// TIA Portal project "Vessel Recycle System 1 Rev1.0" (V14)

(* hardware
DEVICE "S71500/ET200MP station_1"  S7-1500 station
   slot 0: "Rail_0"  Rack  6ES7 590-1***0-0AA0
   slot 0: "PM 70W 120/230VAC"  PM 70W 120/230VAC  6EP1332-4BA00
   slot 1: "PLC_1"  CPU 1511-1 PN  6ES7 511-1AK01-0AB0  V2.0
      slot 3: "CPU display_1"  6ES7591-1AA00-0AA0
DEVICE "ET 200SP station_1"  ET 200SP-Station
   slot 0: "Rack_0"  Rack  6ES5 710-8MAx1
   slot 0: "IO device_1"  IM 155-6 PN BA  6ES7 155-6AR00-0AN0  V3.2
   slot 1: "DI 8x24VDC BA_1"  DI 8x24VDC BA  6ES7 131-6BF00-0AA0  V1.0
      slot 1: "DI 8x24VDC BA_1"  DI 8x24VDC BA
   slot 2: "DI 8x24VDC BA_2"  DI 8x24VDC BA  6ES7 131-6BF00-0AA0  V1.0
      slot 1: "DI 8x24VDC BA_2"  DI 8x24VDC BA
   slot 3: "DQ 8x24VDC/0.5A BA_1"  DQ 8x24VDC/0.5A BA  6ES7 132-6BF00-0AA0  V1.0
      slot 1: "DQ 8x24VDC/0.5A BA_1"  DQ 8x24VDC/0.5A BA
   slot 4: "DQ 8x24VDC/0.5A BA_2"  DQ 8x24VDC/0.5A BA  6ES7 132-6BF00-0AA0  V1.0
      slot 1: "DQ 8x24VDC/0.5A BA_2"  DQ 8x24VDC/0.5A BA
   slot 5: "DQ 8x24VDC/0.5A BA_3"  DQ 8x24VDC/0.5A BA  6ES7 132-6BF00-0AA0  V1.0
      slot 1: "DQ 8x24VDC/0.5A BA_3"  DQ 8x24VDC/0.5A BA
   slot 6: "Server module_1"  Server module  6ES7 193-6PA00-0AA0  V1.1
      slot 1: "Server module_1"  Server module
   slot 127: "BA 2xRJ45"  BA 2xRJ45  6ES7 193-6AR00-0AA0  V0.0
      slot 1: "Port_1"  6ES7 193-6AR00-0AA0  V0.0
      slot 2: "Port_2"  6ES7 193-6AR00-0AA0  V0.0
DEVICE "SCALANCE XB-200"  SCALANCE X-Station
   slot 0: "SCALANCE X rack"  Rail
   slot 0: "Switch_1"  SCALANCE XB208  6GK5 208-0BA00-2AB2  V1.2
DEVICE "HMI_1"  TP1200 Comfort
   slot 0: "TP1200 Comfort"  TP1200 Comfort  6AV2 124-0MC01-0AX0  14.0.0.0
   slot 1: "HMI_RT_1"  TP1200 Comfort  6AV2 124-0MC01-0AX0  14.0.0.0
   slot 5: "HMI_1.IE_CP_1"  PROFINET Interface  14.0.0.0
      slot 1: "PROFINET Interface_1"  PROFINET Interface
         slot 1: "Port_1"  Port
         slot 2: "Port_2"  Port
   slot 7: "HMI_1.MPI/DP_CP_1"  MPI/DP Interface  14.0.0.0
DEVICE "GSD device_1"  GSD.Device.PN
   slot 0: "Rack"  Rack  V1.0
   slot 0: "vr1pump1"  Standard, no PDev  6GK1 953-0CA00  Z1.0
      slot 0: "Standard, no PDev"  Standard, no PDev
      slot 1: "Interface"  Interface
         slot 1: "Port_1"  Port
   slot 1: " 128 bytes I_1"  128 bytes I  1.0
      slot 0: " 128 bytes I"  128 bytes I
   slot 2: " 128 bytes O_1"  128 bytes O  1.0
      slot 0: " 128 bytes O"  128 bytes O
DEVICE "GSD device_2"  GSD.Device.PN
   slot 0: "Rack"  Rack  V1.0
   slot 0: "vr1pump2"  Standard, no PDev  6GK1 953-0CA00  Z1.0
      slot 0: "Standard, no PDev"  Standard, no PDev
      slot 1: "Interface"  Interface
         slot 1: "Port_1"  Port
   slot 1: " 128 bytes I_1"  128 bytes I  1.0
      slot 0: " 128 bytes I"  128 bytes I
   slot 2: " 128 bytes O_1"  128 bytes O  1.0
      slot 0: " 128 bytes O"  128 bytes O
*)

// ===== PLC "PLC_1"  CPU 1511-1 PN =====

VAR_GLOBAL   // PLC tag table "Default tag table"
   "System_Byte" AT %MB1 : Byte;
   "FirstScan" AT %M1.0 : Bool;
   "DiagStatusUpdate" AT %M1.1 : Bool;
   "AlwaysTRUE" AT %M1.2 : Bool;
   "AlwaysFALSE" AT %M1.3 : Bool;
   "Clock_Byte" AT %MB0 : Byte;
   "Clock_10Hz" AT %M0.0 : Bool;
   "Clock_5Hz" AT %M0.1 : Bool;
   "Clock_2.5Hz" AT %M0.2 : Bool;
   "Clock_2Hz" AT %M0.3 : Bool;
   "Clock_1.25Hz" AT %M0.4 : Bool;
   "Clock_1Hz" AT %M0.5 : Bool;
   "Clock_0.625Hz" AT %M0.6 : Bool;
   "Clock_0.5Hz" AT %M0.7 : Bool;
END_VAR

VAR_GLOBAL   // PLC tag table "General Tags"
   "Safety_Relay_Trip" AT %I0.0 : Bool;
   "spare_%I0.3" AT %I0.3 : Bool;
   "UM_HI_Level_SW" AT %I0.6 : Bool;
   "spare_%I0.7" AT %I0.7 : Bool;
   "spare_%Q0.0" AT %Q0.0 : Bool;
   "spare_%Q0.1" AT %Q0.1 : Bool;
   "spare_%Q2.2" AT %Q2.2 : Bool;
   "Buzzer" AT %Q2.5 : Bool;
   "Green_Light" AT %Q2.6 : Bool;
   "Red_Light" AT %Q2.7 : Bool;
   "spare_%Q1.2" AT %Q1.2 : Bool;
   "spare_%Q1.3" AT %Q1.3 : Bool;
   "spare_%Q1.4" AT %Q1.4 : Bool;
   "spare_%Q1.5" AT %Q1.5 : Bool;
   "spare_%Q1.6" AT %Q1.6 : Bool;
   "spare_%Q1.7" AT %Q1.7 : Bool;
   "spare_%I1.6" AT %I1.6 : Bool;
   "spare_%I1.7" AT %I1.7 : Bool;
   "spare_%Q0.2" AT %Q0.2 : Bool;
   "spare_%Q0.3" AT %Q0.3 : Bool;
END_VAR

VAR_GLOBAL   // PLC tag table "Station 1"
   "S1_Start_PB" AT %I0.1 : Bool;
   "S1_Stop_PB" AT %I0.2 : Bool;
   "Safety_Lock1_Engaged" AT %I1.0 : Bool;
   "Safety_Key1_Inserted" AT %I1.1 : Bool;
   "Estop1_PB_Active" AT %I1.4 : Bool;
   "S1_Valve" AT %Q0.4 : Bool;
   "Safety_Lock1_Open" AT %Q0.5 : Bool;
   "Pmp1_Permissive" AT %Q1.0 : Bool;
   "S1_Start_Light" AT %Q2.0 : Bool;
   "S1_Stop_Light" AT %Q2.1 : Bool;
END_VAR

VAR_GLOBAL   // PLC tag table "Station 2"
   "S2_Start_PB" AT %I0.4 : Bool;
   "S2_Stop_PB" AT %I0.5 : Bool;
   "Safety_Lock2_Engaged" AT %I1.2 : Bool;
   "Safety_Key2_Inserted" AT %I1.3 : Bool;
   "Estop2_PB_Active" AT %I1.5 : Bool;
   "S2_Valve" AT %Q0.6 : Bool;
   "Safety_Lock2_Open" AT %Q0.7 : Bool;
   "Pmp2_Permissive" AT %Q1.1 : Bool;
   "S2_Start_Light" AT %Q2.3 : Bool;
   "S2_Stop_Light" AT %Q2.4 : Bool;
END_VAR

TYPE "UDT_MDrive_PQW"
   STRUCT
      Acc : UDInt;   // A
      Dec : UDInt;   // D
      TS : UDInt;   // TS
      V_Init : UDInt;   // VI
      V_Max : UDInt;   // VM
      C1 : DInt;   // C1
      C2 : DInt;   // C2
      HT : DInt;   // HT
      MoveABS : DInt;   // MA
      MoveRel : DInt;   // MR
      Slew : DInt;   // SL
      SetPosition : DInt;   // P
      MT : DInt;   // MT
      MS : UInt;   // MS
      SetError : UInt;   // ER
      AO : UInt;   // AO
      AS : USInt;   // AS
      HC : USInt;   // HC
      OT : USInt;   // OT
      RC : USInt;   // RC
      TQ : USInt;   // TQ
      HM : USInt;   // HM
      HI : USInt;   // HI
      DriveEnable : USInt;   // DriveEnable
      EncoderEnable : USInt;   // EncoderEnable
      TD : USInt;   // TD
      Esc : USInt;   // Esc
      CF : USInt;   // CF
      R9_R10 : Struct
         Reg9 : Bool;
         Bit1 : Bool;
         Bit2 : Bool;
         Bit3 : Bool;
         Bit4 : Bool;
         Bit5 : Bool;
         Bit6 : Bool;
         Bit7 : Bool;
         Reg10 : Bool;
         Bit8 : Bool;
         Bit9 : Bool;
         Bit10 : Bool;
         Bit11 : Bool;
         Bit12 : Bool;
         Bit13 : Bool;
         Bit14 : Bool;
      END_STRUCT;
      R11 : Struct
         Reg11 : Bool;
         Bit1 : Bool;
         Bit2 : Bool;
         Bit3 : Bool;
         Bit4 : Bool;
         Bit5 : Bool;
         Bit6 : Bool;
         Bit7 : Bool;
      END_STRUCT;
      Unused_1 : String[28];
      R1_R38 : Struct
         Dummy_Bit0 : Bool;
         Dummy_Bit1 : Bool;
         Dummy_Bit2 : Bool;
         Dummy_Bit3 : Bool;
         Dummy_Bit4 : Bool;
         Dummy_Bit5 : Bool;
         Dummy_Bit6 : Bool;
         Dummy_Bit7 : Bool;
         Reg1 : Bool;
         Reg2 : Bool;
         Reg3 : Bool;
         Reg4 : Bool;
         Reg5 : Bool;
         Reg6 : Bool;
         Reg7 : Bool;
         Reg8 : Bool;
         Reg9 : Bool;
         Reg10 : Bool;
         Reg11 : Bool;
         Reg12 : Bool;
         Reg13 : Bool;
         Reg14 : Bool;
         Reg15 : Bool;
         Reg16 : Bool;
         Reg17 : Bool;
         Reg18 : Bool;
         Reg19 : Bool;
         Reg20 : Bool;
         Reg21 : Bool;
         Reg22 : Bool;
         Reg23 : Bool;
         Reg24 : Bool;
         Reg25 : Bool;
         Reg26 : Bool;
         Reg27 : Bool;
         Reg28 : Bool;
         Reg32 : Bool;
         Reg33 : Bool;
         Reg38 : Bool;
         Dummy_Bit8 : Bool;
         Dummy_Bit9 : Bool;
         Dummy_Bit10 : Bool;
         Dummy_Bit11 : Bool;
         Dummy_Bit12 : Bool;
         Dummy_Bit13 : Bool;
         Dummy_Bit14 : Bool;
         Dummy_Bit15 : Bool;
         Dummy_Bit16 : Bool;
      END_STRUCT;
      Unused_2 : Array[0..17] of Byte;
   END_STRUCT;
END_TYPE

TYPE "UDT_MDrive_PIW"
   STRUCT
      Acc : UDInt;   // A
      Dec : UDInt;   // D
      TS : UDInt;   // TS
      V_Init : UDInt;   // VI
      V_Max : UDInt;   // VM
      C1 : DInt;   // C1
      C2 : DInt;   // C2
      LL : DInt;   // LL
      V : DInt;   // V
      PC : DInt;   // PC
      MS : DInt;   // MS
      Position : DInt;   // P
      AO : UInt;   // AO
      Dummy_Int : UInt;   // Dummy_Int
      AF : UInt;   // AF
      Error : UInt;   // ER
      I5 : UInt;   // I5
      AS : USInt;   // AS
      HC : USInt;   // HC
      Inputs : USInt;   // IN
      RC : USInt;   // RC
      TQ : USInt;   // TQ
      "OF" : USInt;   // OF
      TE : USInt;   // TE
      DriveEnable : USInt;   // DriveEnable
      EncoderEnable : USInt;   // EncoderEnable
      TD : USInt;   // TD
      MV : USInt;   // MV
      MP : USInt;   // MP
      VC : USInt;   // VC
      ST : USInt;   // ST
      LR : USInt;   // LR
      Dummy_Byte : USInt;
      Unused : Array[0..52] of Byte;
   END_STRUCT;
END_TYPE

TYPE "UDT_MDrive_Data"
   STRUCT
      Target_Position : DInt;   // Input
      Current_Position : DInt := 0;   // Output
      Slew : Struct   // Input
         Fwd : Bool;   // Input
         Rev : Bool;   // Input
         Speed : Real;   // Input
      END_STRUCT;
      State : Struct   // Output
         IsMoving : Bool;   // Output
         IsHomed : Bool;   // Output
         OnPosition : Bool;   // Output
      END_STRUCT;
      ErrorCode : UInt;   // Output
      Inputs : Array[0..7] of Bool;   // Output
      HomeSensor : Bool;   // Output
      Reset : Bool;   // Output
      CMD_Trigger : Struct   // Input
         MoveAbs : Bool;   // Trigger new MA command
         MoveRel : Bool;   // Trigger new MR command
         Slew : Bool;   // Trigger new SL command
         Homing : Bool;   // Trigger new HM command ( Homing )
         SetPos : Bool;   // Trigger new Position
      END_STRUCT;
      CMD_Busy : Bool;   // Output
   END_STRUCT;
END_TYPE

TYPE "UDT_MDrive_Settings"
   STRUCT
      ScaleMax : DInt;
      ScaleMin : DInt;
      MaxSpeed : DInt;
      MinSpeed : DInt;
   END_STRUCT;
END_TYPE

TYPE "UDT_HMI_MDrive"
   STRUCT
      Slew : Struct   // Input
         Fwd : Bool;   // Input
         Rev : Bool;   // Input
         Speed : Real;   // Input
      END_STRUCT;
      State : Struct   // Output
         IsMoving : Bool;   // Output
         IsHomed : Bool;   // Output
         OnPosition : Bool;   // Output
      END_STRUCT;
      Drive_State : USInt;   // Output
      ErrorCode : UInt;   // Output
   END_STRUCT;
END_TYPE

DATA_BLOCK "Setup_Data"   // DB2
{ S7_Optimized_Access := 'TRUE' }
VERSION : 0.1
   VAR
      Estop_Active : Bool;
      Buzzer_Reset : Bool;
   END_VAR
   VAR RETAIN
      Total_Waste_Drum_Volume : Real;
      Waste_Drum_Volume : Real := 100.0;
      Waste_Drum_Percent_Volume : Real;
   END_VAR
   VAR
      Waste_Container_Reset : Bool;
      Waste_Container_Interlock : Bool;
      Waste_Container_Alarm_Level : Int := 0;
      Waste_Container_Alarm_SP : Real := 80.0;
      Waste_Container_Interlock_Level : Real := 90.0;
      Waste_Rad_Level : Real;
   END_VAR
   VAR RETAIN
      Waste_Rad_High_Alarm : Real := 100.0;
   END_VAR
   VAR
      Waste_Rad_Alarm : Bool;
   END_VAR
   VAR RETAIN
      System_Version : String := 'VRS1 Ver 1.0';
   END_VAR
BEGIN
END_DATA_BLOCK

DATA_BLOCK "Discrete_Alarm_Source_DB"   // DB20
{ S7_Optimized_Access := 'TRUE' }
VERSION : 0.1
// stored: InstanceOfName Discrete_Alarm_Source
"Discrete_Alarm_Source"
BEGIN
END_DATA_BLOCK

// folder: Station 1 Data Blocks

DATA_BLOCK "S1_HMI_DB"   // DB1
{ S7_Optimized_Access := 'TRUE' }
VERSION : 0.1
// stored: InstanceOfName Station_HMI
"Station_HMI"
BEGIN
END_DATA_BLOCK

DATA_BLOCK "S1_Auto_Mode_Setpoints"   // DB3
{ S7_Optimized_Access := 'TRUE' }
VERSION : 0.1
   VAR RETAIN
      Pump_Remove_Full_Speed : Real := 300.0;
      Ramp_Remove_Step : Int := 1;
      Ramp_Remove_Time : Time := T#500MS;
      Pump_Drain_Full_Speed : Real := 475.0;
      Ramp_Drain_Step : Int := 1;
      Ramp_Drain_Time : Time := T#500MS;
      Pump_Rinse_Full_Speed : Real := 425.0;
      Ramp_Rinse_Step : Int := 1;
      Ramp_Rinse_Time : Time := T#500MS;
      Run_Remove_Time : Time := T#1M_3S;
      Run_Drain_Time : Time := T#27S;
      Run_Rinse_Time : Time := T#19S;
      Number_of_Rinses : Int := 3;
      Use_RAD_CTRL : Bool := FALSE;
      Rinse_to_RAD_Level : Real := 50.0;
   END_VAR
BEGIN
END_DATA_BLOCK

DATA_BLOCK "S1_General_Setup"   // DB6
{ S7_Optimized_Access := 'TRUE' }
VERSION : 0.1
   VAR
      Manual_Mode : Bool;
      MM_Run_Enable : Bool;
      Auto_Run_Enable : Bool;
      Man_Speed_SP : Real;
      MM_Pump_Slew_PB : Bool;
      MM_Pump_Dir_SW_FWD : Bool;
      MM_Pump_Dir_SW_REV : Bool;
      MM_Valve_Dir_SW : Bool;
      MM_Feedback_RPM : Real;
      Auto_Process_Complete : Bool;
      Auto_Process_Complete_Trig : Bool;
      Manual_Mode_Permissive : Bool;
      Door_Lock_Bypass : Bool;
      Water_Supply_Interlock : Bool;
      Pump_Encoder_Run : Bool;
      Vessel_Rad_Level : Real;
   END_VAR
   VAR RETAIN
      Vessel_Alarm_Level : Real := 100.0;
   END_VAR
   VAR
      Pump_Rad_Level : Real;
   END_VAR
   VAR RETAIN
      Pump_Alarm_Level : Real := 100.0;
   END_VAR
   VAR
      Rad_Lock_Bypass : Bool;
      Rad_Lock : Bool;
   END_VAR
   VAR RETAIN
      Leave_Manual_Screen : Bool;
      Container_Water_Supply_Volume : Real := 3.0;
      Total_Water_Supply_Volume : Real;
      Total_from_Water_Supply_Volume : Real;
      Water_Supply_Interlock_Level : Real := 3.0;
   END_VAR
   VAR
      Total_Water_Supply_Percent : Real;
   END_VAR
   VAR RETAIN
      Total_to_Waste_Volume : Real;
   END_VAR
   VAR
      Pump_Factor : Real := 1.0;
      Pump_Stroke_Volume : Real := 0.192;
      Water_Supply_Alarm_Level : Int;
      Water_Supply_Alarm_SP : Real := 20.0;
      MM_Pump_Feedback : Real;
      Auto_Pump_Feedback_Vel : Real;
      Auto_Pump_Feedback_En : DInt;
      Auto_Pump_Running : Bool;
      Pump_Feedback : Real;
      New_Waste_Container : Bool;
      New_Water_Container : Bool;
      Level_Interlock : Bool;
      Pump_Error_Code : UInt;
      Pump_Error_Bit : Bool;
      MM_Pump_Error_Code : UInt;
      MM_Pump_Error_Bit : Bool;
   END_VAR
BEGIN
END_DATA_BLOCK

DATA_BLOCK "S1_Automated_Run_DB"   // DB7
{ S7_Optimized_Access := 'TRUE' }
VERSION : 0.1
// stored: InstanceOfName Automated_Run
"Automated_Run"
BEGIN
END_DATA_BLOCK

DATA_BLOCK "S1_ Door_Lock_Control_DB"   // DB9
{ S7_Optimized_Access := 'TRUE' }
VERSION : 0.1
// stored: InstanceOfName Door_Lock_Control
"Door_Lock_Control"
BEGIN
END_DATA_BLOCK

DATA_BLOCK "S1_Interlocks_DB"   // DB10
{ S7_Optimized_Access := 'TRUE' }
VERSION : 0.1
// stored: InstanceOfName Interlocks
"Interlocks"
BEGIN
END_DATA_BLOCK

DATA_BLOCK "Manual_Run_S1_DB"   // DB23
{ S7_Optimized_Access := 'TRUE' }
VERSION : 0.1
// stored: InstanceOfName Manual_ Run
"Manual_ Run"
BEGIN
END_DATA_BLOCK

// folder: Station 1 Data Blocks/Pump 1 Data Blocks

DATA_BLOCK "Pmp1_MM_HMI_DB"   // DB5
{ S7_Optimized_Access := 'TRUE' }
VERSION : 0.1
// stored: InstanceOfName Pump_HMI
"Pump_HMI"
BEGIN
END_DATA_BLOCK

DATA_BLOCK "Pmp1_Auto_HMI_DB"   // DB13
{ S7_Optimized_Access := 'TRUE' }
VERSION : 0.1
// stored: InstanceOfName Pump_HMI
"Pump_HMI"
BEGIN
END_DATA_BLOCK

DATA_BLOCK "Pmp1_Settings"   // DB21
{ S7_Optimized_Access := 'TRUE' }
VERSION : 0.1
   VAR RETAIN
      Settings : "UDT_MDrive_Settings";   // 0-100% in 0.1% Steps
   END_VAR
BEGIN
   Settings.ScaleMax := 100;
   Settings.MaxSpeed := 1000000;
END_DATA_BLOCK

DATA_BLOCK "Pmp1_Data"   // DB22
{ S7_Optimized_Access := 'TRUE' }
VERSION : 0.1
   VAR
      Data : "UDT_MDrive_Data";
   END_VAR
BEGIN
END_DATA_BLOCK

DATA_BLOCK "Pmp1_Control_DB"   // DB24
{ S7_Optimized_Access := 'TRUE' }
VERSION : 0.1
// stored: InstanceOfName Motor_Control
"Motor_Control"
BEGIN
END_DATA_BLOCK

// folder: Station 2 Data Blocks

DATA_BLOCK "S2_General_Setup"   // DB4
{ S7_Optimized_Access := 'TRUE' }
VERSION : 0.1
   VAR
      Pump_Alarm_Level : Real := 100.0;
      Pump_Rad_Level : Real;
      Vessel_Alarm_Level : Real := 100.0;
      Vessel_Rad_Level : Real;
      Manual_Mode : Bool;
      Man_Speed_SP : Real;
      MM_Pump_Dir_SW_FWD : Bool;
      MM_Pump_Dir_SW_REV : Bool;
      MM_Pump_Slew_PB : Bool;
      MM_Valve_Dir_SW : Bool;
      MM_Run_Enable : Bool;
      MM_Pump_Feedback : Real;
      MM_Feedback_RPM : Real;
      Water_Supply_Interlock : Bool;
      Door_Lock_Bypass : Bool;
      Rad_Lock_Bypass : Bool;
   END_VAR
   VAR RETAIN
      Leave_Manual_Screen : Bool;
   END_VAR
   VAR
      Rad_Lock : Bool;
      Auto_Process_Complete : Bool;
      Auto_Process_Complete_Trigger : Bool;
      Auto_Run_Enable : Bool;
      Auto_Pump_Running : Bool;
      Pump_Encoder_Run : Bool;
      Auto_Pump_Feedback_Vel : Real;
      Auto_Pump_Feedback_En : DInt;
      Pump_Error_Code : UInt;
      Pump_Error_Bit : Bool;
      Manual_Mode_Permissive : Bool;
   END_VAR
   VAR RETAIN
      Container_Water_Supply_Volume : Real := 3.0;
      Total_Water_Supply_Volume : Real;
   END_VAR
   VAR
      Total_Water_Supply_Percent : Real;
   END_VAR
   VAR RETAIN
      Total_from_Water_Supply_Volume : Real;
      Total_to_Waste_Volume : Real;
   END_VAR
   VAR
      Pump_Factor : Real := 1.0;
      Pump_Stroke_Volume : Real := 0.192;
      Removed_from_Water_Supply : Real;
      Water_Supply_Alarm_Level : Int;
      Water_Supply_Alarm_SP : Real := 20.0;
      New_Waste_Container : Bool;
      New_Water_Container : Bool;
      Level_Interlock : Bool;
   END_VAR
   VAR RETAIN
      Water_Supply_Interlock_Level : Real := 0.0;
   END_VAR
   VAR
      MM_Pump_Error_Code : UInt;
      MM_Pump_Error_Bit : Bool;
   END_VAR
BEGIN
END_DATA_BLOCK

DATA_BLOCK "S2_Auto_Mode_Setpoints"   // DB11
{ S7_Optimized_Access := 'TRUE' }
VERSION : 0.1
   VAR RETAIN
      Pump_Remove_Full_Speed : Real := 425.0;
      Ramp_Remove_Step : Int := 1;
      Ramp_Remove_Time : Time := T#500MS;
      "Pump_Drain_Full Speed" : Real := 600.0;
      Ramp_Drain_Step : Int := 1;
      Ramp_Drain_Time : Time := T#500MS;
      Pump_Rinse_Full_Speed : Real := 500.0;
      Ramp_Rinse_Step : Int := 1;
      Ramp_Rinse_Time : Time := T#500MS;
      Run_Remove_Time : Time := T#55S;
      Run_Drain_Time : Time := T#27S;
      Run_Rinse_Time : Time := T#21S_500MS;
      Number_of_Rinses : Int := 3;
      Use_RAD_CTRL : Bool := FALSE;
      Rinse_to_RAD_Level : Real := 0.0;
   END_VAR
BEGIN
END_DATA_BLOCK

DATA_BLOCK "S2_Automated_Run_DB"   // DB12
{ S7_Optimized_Access := 'TRUE' }
VERSION : 0.1
// stored: InstanceOfName Automated_Run
"Automated_Run"
BEGIN
END_DATA_BLOCK

DATA_BLOCK "S2_Door_Lock_Control_DB"   // DB14
{ S7_Optimized_Access := 'TRUE' }
VERSION : 0.1
// stored: InstanceOfName Door_Lock_Control
"Door_Lock_Control"
BEGIN
END_DATA_BLOCK

DATA_BLOCK "S2_Interlocks_DB"   // DB15
{ S7_Optimized_Access := 'TRUE' }
VERSION : 0.1
// stored: InstanceOfName Interlocks
"Interlocks"
BEGIN
END_DATA_BLOCK

DATA_BLOCK "S2_HMIl_DB"   // DB17
{ S7_Optimized_Access := 'TRUE' }
VERSION : 0.1
// stored: InstanceOfName Station_HMI
"Station_HMI"
BEGIN
END_DATA_BLOCK

DATA_BLOCK "Manual_ Run_S2_DB"   // DB25
{ S7_Optimized_Access := 'TRUE' }
VERSION : 0.1
// stored: InstanceOfName Manual_ Run
"Manual_ Run"
BEGIN
END_DATA_BLOCK

// folder: Station 2 Data Blocks/Pump 2 Data Blocks

DATA_BLOCK "Pmp2_Control_DB"   // DB26
{ S7_Optimized_Access := 'TRUE' }
VERSION : 0.1
// stored: InstanceOfName Motor_Control
"Motor_Control"
BEGIN
END_DATA_BLOCK

DATA_BLOCK "Pmp2_MM_HMI_DB"   // DB27
{ S7_Optimized_Access := 'TRUE' }
VERSION : 0.1
// stored: InstanceOfName Pump_HMI
"Pump_HMI"
BEGIN
END_DATA_BLOCK

DATA_BLOCK "Pmp2_Settings"   // DB28
{ S7_Optimized_Access := 'TRUE' }
VERSION : 0.1
   VAR RETAIN
      Settings : "UDT_MDrive_Settings";   // 0-100% in 0.1% Steps
   END_VAR
BEGIN
   Settings.ScaleMax := 100;
   Settings.MaxSpeed := 1000000;
END_DATA_BLOCK

DATA_BLOCK "Pmp2_Data"   // DB29
{ S7_Optimized_Access := 'TRUE' }
VERSION : 0.1
   VAR
      Data : "UDT_MDrive_Data";
   END_VAR
BEGIN
END_DATA_BLOCK

DATA_BLOCK "Pmp2_Auto_HMI_DB"   // DB30
{ S7_Optimized_Access := 'TRUE' }
VERSION : 0.1
// stored: InstanceOfName Pump_HMI
"Pump_HMI"
BEGIN
END_DATA_BLOCK

// folder: (top level)

FUNCTION_BLOCK "Station_HMI"   // FB1, SCL
{ S7_Optimized_Access := 'TRUE' }
VERSION : 0.1
   VAR_INPUT
      Valve_Direction : Bool;
      MM_Valve_Direction : Bool;
      Pump_Direction_FWD : Bool;
      MM_Pump_Direction_FWD : Bool;
      Pump_Direction_REV : Bool;
      MM_Pump_Direction_REV : Bool;
      Pump_Run : Bool;
      MM_Pump_Run : Bool;
      Manual_Mode : Bool;
      Safety_Key_Inserted : Bool;
      Safety_Lock_Engaged : Bool;
      Process_Complete : Bool;
      Rad_lock : Bool;
      Auto_Use_RAD_CTRL : Bool;
      Total_Water_Supply_Percent : Real;
      Water_Supply_Alarm_SP : Real;
   END_VAR
   VAR_OUTPUT
      Water_Supply_Alarm_Level : Int;
   END_VAR
   VAR
      Valve_Drain : Int;
      Valve_Rinse : Int;
      Valve_Pump : Int;
      Tubing_Rinse : Int;
      Tubing_Pump : Int;
      Tubing_Drain : Int;
      Tubing_Vessel : Int;
      Display_PMP_FWD : Bool;
      Display_PMP_REV : Bool;
      Door_Closed : Int;
      Door_Locked : Bool;
      Hide_Vessel_Tubing : Bool;
      Recycle_Mode_HMI : String;
      Door_Lock_Bypass_HMI : Bool;
      Auto_Info_HMI : Int;
      Warning_1 : Bool;
      Warning_2 : Bool;
   END_VAR
BEGIN

   IF (#Process_Complete=TRUE AND #Rad_lock=FALSE) THEN
       #Door_Lock_Bypass_HMI:=TRUE;
   ELSE
       #Door_Lock_Bypass_HMI := FALSE;
   END_IF;

   IF (#Auto_Use_RAD_CTRL = TRUE) THEN
       #Auto_Info_HMI := 1;
   ELSIF (#Auto_Use_RAD_CTRL = FALSE) THEN
       #Auto_Info_HMI := 2;
   ELSE
       #Auto_Info_HMI := 3;
   END_IF;

   IF #Manual_Mode = False THEN

       #Recycle_Mode_HMI := 'AUTO';
       #Warning_1 := 0;
       #Warning_2 := 0;

       IF (#Valve_Direction = FALSE AND #Pump_Run = TRUE) THEN
           #Valve_Drain := 2;
           #Valve_Pump := 2;
           #Valve_Rinse := 3;
           #Tubing_Pump := 2;
           #Tubing_Drain := 2;
           #Tubing_Rinse := 3;
           #Tubing_Vessel := 2;
       ELSIF (#Valve_Direction = TRUE AND #Pump_Run = TRUE) THEN
           #Valve_Rinse := 1;
           #Valve_Pump := 1;
           #Valve_Drain := 3;
           #Tubing_Pump := 1;
           #Tubing_Rinse := 1;
           #Tubing_Drain := 3;
           #Tubing_Vessel := 1;
       ELSE
           #Valve_Drain := 0;
           #Valve_Rinse := 0;
           #Valve_Pump := 0;
           #Tubing_Pump := 0;
           #Tubing_Rinse := 0;
           #Tubing_Drain := 0;
           #Tubing_Vessel := 0;
       END_IF;

       IF (#Pump_Direction_FWD = TRUE AND #Pump_Direction_REV = FALSE AND #Pump_Run = TRUE) THEN
           #Display_PMP_FWD := TRUE;
           #Display_PMP_REV := FALSE;
       ELSIF (#Pump_Direction_FWD = FALSE AND #Pump_Direction_REV = TRUE AND #Pump_Run = TRUE) THEN
           #Display_PMP_REV := TRUE;
           #Display_PMP_FWD := FALSE;
       ELSE
           #Display_PMP_FWD := FALSE;
           #Display_PMP_REV := FALSE;
       END_IF;

   END_IF;


   IF #Manual_Mode = TRUE THEN

       #Recycle_Mode_HMI := 'MANUAL';

       IF (#MM_Valve_Direction = FALSE AND #MM_Pump_Direction_FWD = TRUE) THEN
           #Warning_1 := 0;
           #Warning_2 := 0;
       ELSIF (#MM_Valve_Direction = FALSE AND #MM_Pump_Direction_REV = TRUE) THEN
           #Warning_1 := 1;
           #Warning_2 := 0;
       ELSIF (#MM_Valve_Direction = TRUE AND #MM_Pump_Direction_FWD = TRUE) THEN
           #Warning_1 := 0;
           #Warning_2 := 1;
       ELSIF (#MM_Valve_Direction = TRUE AND #MM_Pump_Direction_REV = TRUE) THEN
           #Warning_1 := 0;
           #Warning_2 := 0;
       ELSE
           #Warning_1 := 0;
           #Warning_2 := 0;
       END_IF;

       IF (#MM_Valve_Direction = FALSE AND #MM_Pump_Direction_FWD = TRUE AND #MM_Pump_Run = TRUE) THEN
           #Valve_Drain := 2;
           #Valve_Pump := 2;
           #Valve_Rinse := 3;
           #Tubing_Pump := 2;
           #Tubing_Drain := 2;
           #Tubing_Rinse := 3;
           #Tubing_Vessel := 2;
       ELSIF (#MM_Valve_Direction = FALSE AND #MM_Pump_Direction_REV = TRUE AND #MM_Pump_Run = TRUE) THEN
           #Valve_Drain := 2;
           #Valve_Pump := 2;
           #Valve_Rinse := 3;
           #Tubing_Pump := 2;
           #Tubing_Drain := 2;
           #Tubing_Rinse := 3;
           #Tubing_Vessel := 2;
       ELSIF (#MM_Valve_Direction = TRUE AND #MM_Pump_Direction_FWD = TRUE AND #MM_Pump_Run = TRUE) THEN
           #Valve_Rinse := 2;
           #Valve_Pump := 2;
           #Valve_Drain := 3;
           #Tubing_Pump := 2;
           #Tubing_Rinse := 2;
           #Tubing_Drain := 3;
           #Tubing_Vessel := 2;
       ELSIF (#MM_Valve_Direction = TRUE AND #MM_Pump_Direction_REV = TRUE AND #MM_Pump_Run = TRUE) THEN
           #Valve_Rinse := 1;
           #Valve_Pump := 1;
           #Valve_Drain := 3;
           #Tubing_Pump := 1;
           #Tubing_Rinse := 1;
           #Tubing_Drain := 3;
           #Tubing_Vessel := 1;
       ELSE
           #Valve_Drain := 0;
           #Valve_Rinse := 0;
           #Valve_Pump := 0;
           #Tubing_Pump := 0;
           #Tubing_Rinse := 0;
           #Tubing_Drain := 0;
           #Tubing_Vessel := 0;
       END_IF;

       IF (#MM_Pump_Direction_FWD = TRUE AND #MM_Pump_Direction_REV = FALSE AND #MM_Pump_Run = TRUE) THEN
           #Display_PMP_FWD := TRUE;
           #Display_PMP_REV := FALSE;
       ELSIF (#MM_Pump_Direction_FWD = FALSE AND #MM_Pump_Direction_REV = TRUE AND #MM_Pump_Run = TRUE) THEN
           #Display_PMP_REV := TRUE;
           #Display_PMP_FWD := FALSE;
       ELSE
           #Display_PMP_FWD := FALSE;
           #Display_PMP_REV := FALSE;
       END_IF;

   END_IF;

   IF (#Safety_Key_Inserted = TRUE AND #Safety_Lock_Engaged = FALSE) THEN
       #Hide_Vessel_Tubing := TRUE;
   ELSE
       #Hide_Vessel_Tubing := FALSE;
   END_IF;

   IF #Safety_Key_Inserted = TRUE THEN
       #Door_Closed:=50;
   ELSE
       #Door_Closed:=0;
   END_IF;

   IF #Safety_Lock_Engaged = TRUE THEN
       #Door_Locked:=TRUE;
   ELSE
       #Door_Locked := FALSE;
   END_IF;



   IF #Total_Water_Supply_Percent < #Water_Supply_Alarm_SP THEN
       #Water_Supply_Alarm_Level := 2;
   ELSE
       #Water_Supply_Alarm_Level := 1;
   END_IF;
END_FUNCTION_BLOCK

FUNCTION_BLOCK "Automated_Run"   // FB2, LAD
{ S7_Optimized_Access := 'TRUE' }
VERSION : 0.1
// Function Block - Automated Run: Main automatic mode routine
// Called by: Main (OB1)
// Calls: Auto_Mode (FB6) - 2 Instances: S1_Automated_Run_DB (DB7), S2_Automated_Run_DB (DB12)
   VAR_INPUT
      Safety_Lock_Engaged : Bool;
      Start_PB : Bool;
      Stop_PB : Bool;
      Estop_Active : Bool;
      Level_Interlock : Bool;
      UM_HI_Level_Interlock : Bool;
      Auto_Pump_Remove_Full_Speed : Real;
      Auto_Ramp_Remove_Step : Int;
      Auto_Ramp_Remove_Time : Time;
      Auto_Pump_Drain_Full_Speed : Real;
      Auto_Ramp_Drain_Step : Int;
      Auto_Ramp_Drain_Time : Time;
      Auto_Pump_Rinse_Full_Speed : Real;
      Auto_Ramp_Rinse_Step : Int;
      Auto_Ramp_Rinse_Time : Time;
      Auto_Run_Drain_Time : Time;
      Auto_Run_Remove_Time : Time;
      Auto_Run_Rinse_Time : Time;
      Auto_Number_of_Rinses : Int;
      Auto_RAD_CTRL : Bool;
      Pump_Cave_RAD_Level : Real;
      Rinse_to_RAD_Level : Real;
      Pump_Factor : Real;
      Pump_Stroke_Volume : Real;
      Pump_Running : Bool;
      Pump_Run_En : Bool;
   END_VAR
   VAR_OUTPUT
      Start_Light : Bool;
      Stop_Light : Bool;
      Pump_Direction_FWD : Bool;
      Pump_Direction_REV : Bool;
      Pump_Enable : Bool;
      Valve_Direction : Bool;
      Pump_Run : Bool;
      Pump_Speed : Real;
   END_VAR
   VAR_IN_OUT
      Total_Flow_from_Supply : Real;
      Total_Flow_to_Waste : Real;
      Water_Container_Reset : Bool;
      Waste_Container_Reset : Bool;
      Process_Complete : Bool;
   END_VAR
   VAR
      Auto_Current_Process_State : String;
      Auto_Current_Rinse_Number : Int;
      Process_Running : Bool;
      Process_Stop : Bool;
      Pump_Fail : Bool;
      Pump_Fail_Alarm : Bool;
      Start_PB_On : Bool;
      Abort_Stop : Bool;
      Run_State : Int;
      Edge_data_bit_1 : Bool;
      Init_Bit : Bool;
      Auto_Mode_Instance : "Auto_Mode";
      IEC_Timer_0_Instance : TON_TIME;
   END_VAR
   VAR CONSTANT
      INIT : Int := 1;
      RUN : Int := 10;
      STOP : Int := 20;
   END_VAR
   VAR_TEMP   // added for the SCL form of the ladder/FBD networks
      _w1 : Bool;
   END_VAR
BEGIN

REGION Network 1
   // Auto Mode start logic and checks for pump not running failure
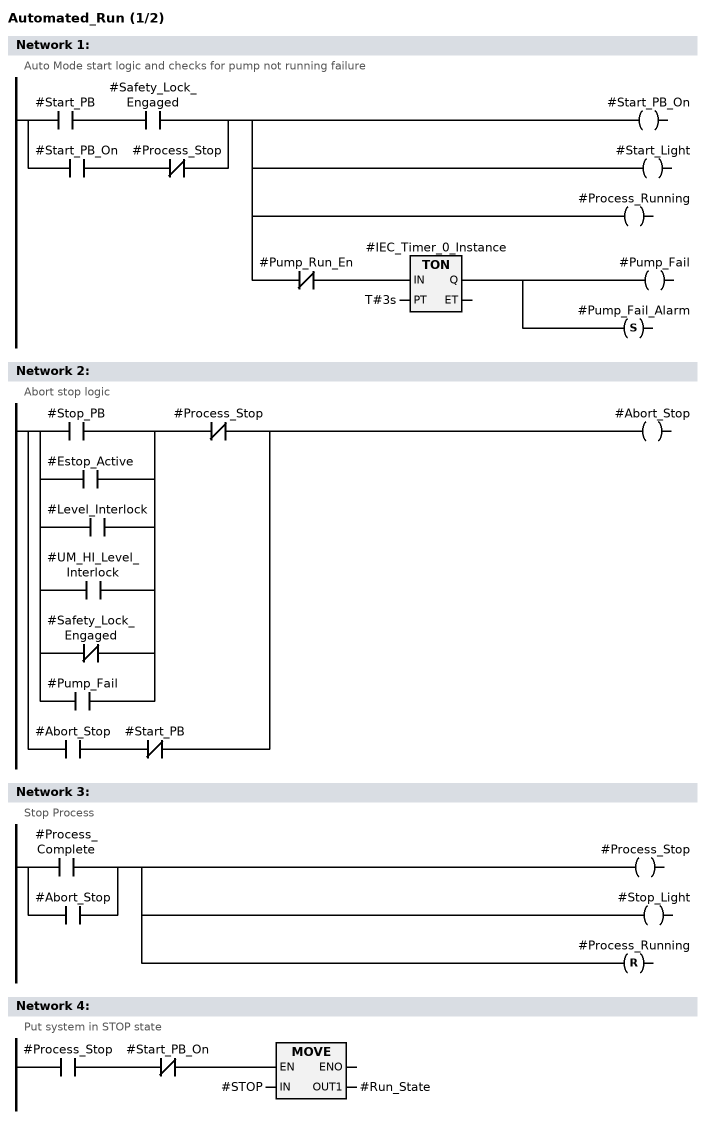
   #Start_PB_On := (#Start_PB AND #Safety_Lock_Engaged) OR (#Start_PB_On AND NOT #Process_Stop);
   #Start_Light := #Start_PB_On;
   #Process_Running := #Start_PB_On;
   #IEC_Timer_0_Instance(IN := #Start_PB_On AND NOT #Pump_Run_En, PT := T#3s);   // TON
   #Pump_Fail := #IEC_Timer_0_Instance.Q;
   IF #IEC_Timer_0_Instance.Q THEN #Pump_Fail_Alarm := TRUE; END_IF;
END_REGION

REGION Network 2
   // Abort stop logic
   RUNG wire#powerrail
      Contact( #Stop_PB )
      wire#w1
      I_Contact( #Process_Stop )
      wire#w2
      Coil( #Abort_Stop )
   END_RUNG
   RUNG wire#powerrail
      Contact( #Estop_Active )
   END_RUNG wire#w1
   RUNG wire#powerrail
      Contact( #Level_Interlock )
   END_RUNG wire#w1
   RUNG wire#powerrail
      Contact( #UM_HI_Level_Interlock )
   END_RUNG wire#w1
   RUNG wire#powerrail
      I_Contact( #Safety_Lock_Engaged )
   END_RUNG wire#w1
   RUNG wire#powerrail
      Contact( #Pump_Fail )
   END_RUNG wire#w1
   RUNG wire#powerrail
      Contact( #Abort_Stop )
      I_Contact( #Start_PB )
   END_RUNG wire#w2
   // the same network as SCL:
   #Abort_Stop := ((#Stop_PB OR #Estop_Active OR #Level_Interlock OR #UM_HI_Level_Interlock OR NOT #Safety_Lock_Engaged OR #Pump_Fail) AND NOT #Process_Stop) OR (#Abort_Stop AND NOT #Start_PB);
END_REGION

REGION Network 3
   // Stop Process
   RUNG wire#powerrail
      Contact( #Process_Complete )
      wire#w1
      Coil( #Process_Stop )
   END_RUNG
   RUNG wire#powerrail
      Contact( #Abort_Stop )
   END_RUNG wire#w1
   RUNG wire#w1
      Coil( #Stop_Light )
   END_RUNG
   RUNG wire#w1
      R_Coil( #Process_Running )
   END_RUNG
   // the same network as SCL:
   #Process_Stop := #Process_Complete OR #Abort_Stop;
   #Stop_Light := #Process_Stop;
   IF #Process_Stop THEN #Process_Running := FALSE; END_IF;
END_REGION

REGION Network 4
   // Put system in STOP state
   RUNG wire#powerrail
      Contact( #Process_Stop )
      I_Contact( #Start_PB_On )
      Move(in := #STOP, out1 => #Run_State)
   END_RUNG
   // the same network as SCL:
   IF #Process_Stop AND NOT #Start_PB_On THEN #Run_State := #STOP; END_IF;
END_REGION

REGION Network 5
   // Put system in INIT state
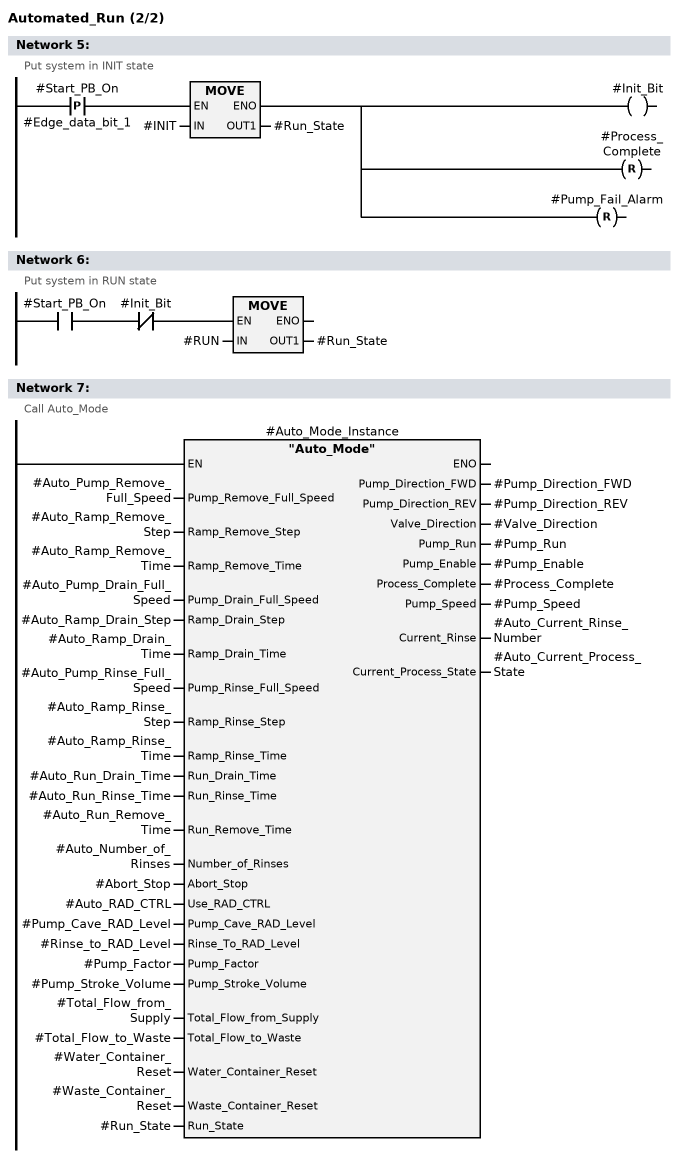
   RUNG wire#powerrail
      P_Contact(operand := #Start_PB_On, bit := #Edge_data_bit_1)
      Move(in := #INIT, out1 => #Run_State)
      wire#w1
      Coil( #Init_Bit )
   END_RUNG
   RUNG wire#w1
      R_Coil( #Process_Complete )
   END_RUNG
   RUNG wire#w1
      R_Coil( #Pump_Fail_Alarm )
   END_RUNG
   // the same network as SCL:
   #_w1 := #Start_PB_On AND NOT #Edge_data_bit_1;   // rising edge of #Start_PB_On
   #Edge_data_bit_1 := #Start_PB_On;
   IF #_w1 THEN #Run_State := #INIT; END_IF;
   #Init_Bit := #_w1;
   IF #_w1 THEN
       #Process_Complete := FALSE;
       #Pump_Fail_Alarm := FALSE;
   END_IF;
END_REGION

REGION Network 6
   // Put system in RUN state
   RUNG wire#powerrail
      Contact( #Start_PB_On )
      I_Contact( #Init_Bit )
      Move(in := #RUN, out1 => #Run_State)
   END_RUNG
   // the same network as SCL:
   IF #Start_PB_On AND NOT #Init_Bit THEN #Run_State := #RUN; END_IF;
END_REGION

REGION Network 7
   // Call Auto_Mode
   RUNG wire#powerrail
      #Auto_Mode_Instance(Pump_Remove_Full_Speed := #Auto_Pump_Remove_Full_Speed, Ramp_Remove_Step := #Auto_Ramp_Remove_Step, Ramp_Remove_Time := #Auto_Ramp_Remove_Time, Pump_Drain_Full_Speed := #Auto_Pump_Drain_Full_Speed, Ramp_Drain_Step := #Auto_Ramp_Drain_Step, Ramp_Drain_Time := #Auto_Ramp_Drain_Time, Pump_Rinse_Full_Speed := #Auto_Pump_Rinse_Full_Speed, Ramp_Rinse_Step := #Auto_Ramp_Rinse_Step, Ramp_Rinse_Time := #Auto_Ramp_Rinse_Time, Run_Drain_Time := #Auto_Run_Drain_Time, Run_Rinse_Time := #Auto_Run_Rinse_Time, Run_Remove_Time := #Auto_Run_Remove_Time, Number_of_Rinses := #Auto_Number_of_Rinses, Abort_Stop := #Abort_Stop, Use_RAD_CTRL := #Auto_RAD_CTRL, Pump_Cave_RAD_Level := #Pump_Cave_RAD_Level, Rinse_To_RAD_Level := #Rinse_to_RAD_Level, Pump_Factor := #Pump_Factor, Pump_Stroke_Volume := #Pump_Stroke_Volume, Total_Flow_from_Supply := #Total_Flow_from_Supply, Total_Flow_to_Waste := #Total_Flow_to_Waste, Water_Container_Reset := #Water_Container_Reset, Waste_Container_Reset := #Waste_Container_Reset, Run_State := #Run_State, Pump_Direction_FWD => #Pump_Direction_FWD, Pump_Direction_REV => #Pump_Direction_REV, Valve_Direction => #Valve_Direction, Pump_Run => #Pump_Run, Pump_Enable => #Pump_Enable, Process_Complete => #Process_Complete, Pump_Speed => #Pump_Speed, Current_Rinse => #Auto_Current_Rinse_Number, Current_Process_State => #Auto_Current_Process_State)
   END_RUNG
   // the same network as SCL:
   #Auto_Mode_Instance(Pump_Remove_Full_Speed := #Auto_Pump_Remove_Full_Speed,   // "Auto_Mode"
                       Ramp_Remove_Step := #Auto_Ramp_Remove_Step,
                       Ramp_Remove_Time := #Auto_Ramp_Remove_Time,
                       Pump_Drain_Full_Speed := #Auto_Pump_Drain_Full_Speed,
                       Ramp_Drain_Step := #Auto_Ramp_Drain_Step,
                       Ramp_Drain_Time := #Auto_Ramp_Drain_Time,
                       Pump_Rinse_Full_Speed := #Auto_Pump_Rinse_Full_Speed,
                       Ramp_Rinse_Step := #Auto_Ramp_Rinse_Step,
                       Ramp_Rinse_Time := #Auto_Ramp_Rinse_Time,
                       Run_Drain_Time := #Auto_Run_Drain_Time,
                       Run_Rinse_Time := #Auto_Run_Rinse_Time,
                       Run_Remove_Time := #Auto_Run_Remove_Time,
                       Number_of_Rinses := #Auto_Number_of_Rinses,
                       Abort_Stop := #Abort_Stop,
                       Use_RAD_CTRL := #Auto_RAD_CTRL,
                       Pump_Cave_RAD_Level := #Pump_Cave_RAD_Level,
                       Rinse_To_RAD_Level := #Rinse_to_RAD_Level,
                       Pump_Factor := #Pump_Factor,
                       Pump_Stroke_Volume := #Pump_Stroke_Volume,
                       Total_Flow_from_Supply := #Total_Flow_from_Supply,
                       Total_Flow_to_Waste := #Total_Flow_to_Waste,
                       Water_Container_Reset := #Water_Container_Reset,
                       Waste_Container_Reset := #Waste_Container_Reset,
                       Run_State := #Run_State,
                       Pump_Direction_FWD => #Pump_Direction_FWD,
                       Pump_Direction_REV => #Pump_Direction_REV,
                       Valve_Direction => #Valve_Direction,
                       Pump_Run => #Pump_Run,
                       Pump_Enable => #Pump_Enable,
                       Process_Complete => #Process_Complete,
                       Pump_Speed => #Pump_Speed,
                       Current_Rinse => #Auto_Current_Rinse_Number,
                       Current_Process_State => #Auto_Current_Process_State);
END_REGION
END_FUNCTION_BLOCK

FUNCTION_BLOCK "Manual_ Run"   // FB3, LAD
{ S7_Optimized_Access := 'TRUE' }
VERSION : 0.1
   VAR_INPUT
      Pump_Permissive : Bool;
      Leave_Manual_Screen : Bool;
      Estop_Active : Bool;
   END_VAR
   VAR_OUTPUT
      Valve_Direction : Bool;
      Pump_Run : Bool;
      Pump_Dir_REV : Bool;
      Pump_Dir_FWD : Bool;
      Pump_Speed_Counts : Real;
      Pump_Run_Enable : Bool;
   END_VAR
   VAR_IN_OUT
      Pump_SP : Real;
      Manual_Mode : Bool;
      Valve_Direction_SW : Bool;
      Pump_Dir_SW_FWD : Bool;
      Pump_Dir_SW_REV : Bool;
      Pump_Run_PB_Slew : Bool;
   END_VAR
   VAR
      Enable : Bool;
   END_VAR
   VAR_TEMP   // added for the SCL form of the ladder/FBD networks
      _w1 : Bool;
   END_VAR
BEGIN

REGION Network 1
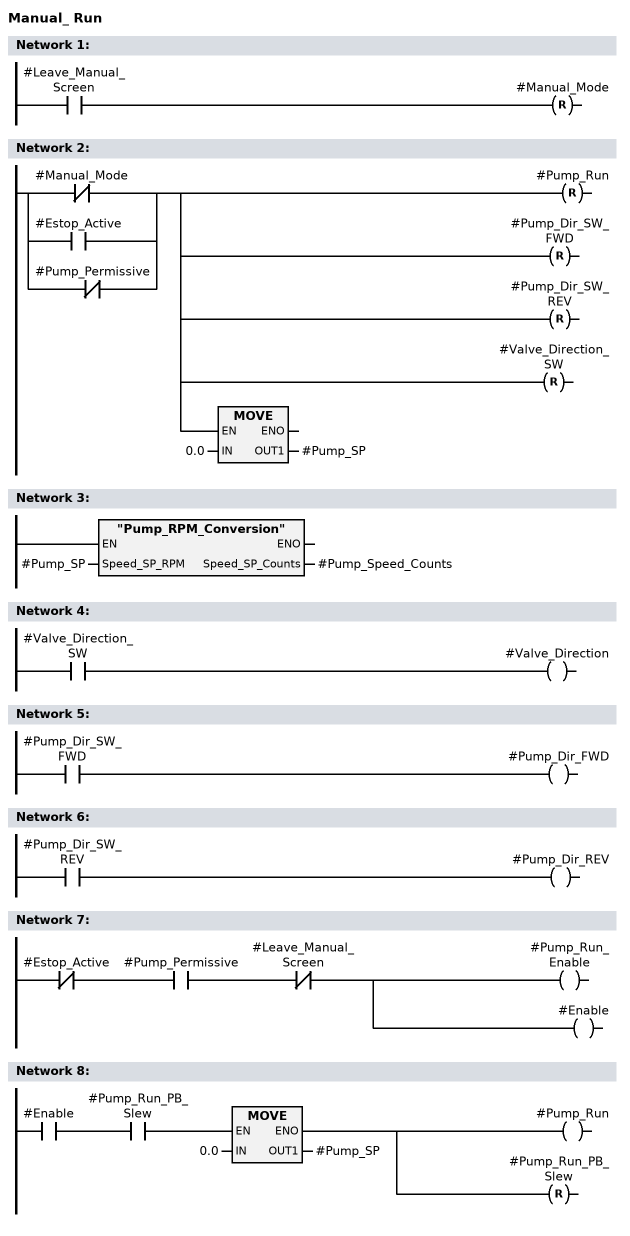
   RUNG wire#powerrail
      Contact( #Leave_Manual_Screen )
      R_Coil( #Manual_Mode )
   END_RUNG
   // the same network as SCL:
   IF #Leave_Manual_Screen THEN #Manual_Mode := FALSE; END_IF;
END_REGION

REGION Network 2
   RUNG wire#powerrail
      I_Contact( #Manual_Mode )
      wire#w1
      R_Coil( #Pump_Run )
   END_RUNG
   RUNG wire#powerrail
      Contact( #Estop_Active )
   END_RUNG wire#w1
   RUNG wire#powerrail
      I_Contact( #Pump_Permissive )
   END_RUNG wire#w1
   RUNG wire#w1
      R_Coil( #Pump_Dir_SW_FWD )
   END_RUNG
   RUNG wire#w1
      R_Coil( #Pump_Dir_SW_REV )
   END_RUNG
   RUNG wire#w1
      R_Coil( #Valve_Direction_SW )
   END_RUNG
   RUNG wire#w1
      Move(in := 0.0, out1 => #Pump_SP)
   END_RUNG
   // the same network as SCL:
   IF NOT #Manual_Mode OR #Estop_Active OR NOT #Pump_Permissive THEN
       #Pump_Run := FALSE;
       #Pump_Dir_SW_FWD := FALSE;
       #Pump_Dir_SW_REV := FALSE;
       #Valve_Direction_SW := FALSE;
       #Pump_SP := 0.0;
   END_IF;
END_REGION

REGION Network 3
   RUNG wire#powerrail
      "Pump_RPM_Conversion"(Speed_SP_RPM := #Pump_SP, Speed_SP_Counts => #Pump_Speed_Counts)
   END_RUNG
   // the same network as SCL:
   "Pump_RPM_Conversion"(Speed_SP_RPM := #Pump_SP, Speed_SP_Counts => #Pump_Speed_Counts);
END_REGION

REGION Network 4
   RUNG wire#powerrail
      Contact( #Valve_Direction_SW )
      Coil( #Valve_Direction )
   END_RUNG
   // the same network as SCL:
   #Valve_Direction := #Valve_Direction_SW;
END_REGION

REGION Network 5
   RUNG wire#powerrail
      Contact( #Pump_Dir_SW_FWD )
      Coil( #Pump_Dir_FWD )
   END_RUNG
   // the same network as SCL:
   #Pump_Dir_FWD := #Pump_Dir_SW_FWD;
END_REGION

REGION Network 6
   RUNG wire#powerrail
      Contact( #Pump_Dir_SW_REV )
      Coil( #Pump_Dir_REV )
   END_RUNG
   // the same network as SCL:
   #Pump_Dir_REV := #Pump_Dir_SW_REV;
END_REGION

REGION Network 7
   RUNG wire#powerrail
      I_Contact( #Estop_Active )
      Contact( #Pump_Permissive )
      I_Contact( #Leave_Manual_Screen )
      wire#w1
      Coil( #Pump_Run_Enable )
   END_RUNG
   RUNG wire#w1
      Coil( #Enable )
   END_RUNG
   // the same network as SCL:
   #Pump_Run_Enable := NOT #Estop_Active AND #Pump_Permissive AND NOT #Leave_Manual_Screen;
   #Enable := #Pump_Run_Enable;
END_REGION

REGION Network 8
   RUNG wire#powerrail
      Contact( #Enable )
      Contact( #Pump_Run_PB_Slew )
      Move(in := 0.0, out1 => #Pump_SP)
      wire#w1
      Coil( #Pump_Run )
   END_RUNG
   RUNG wire#w1
      R_Coil( #Pump_Run_PB_Slew )
   END_RUNG
   // the same network as SCL:
   #_w1 := #Enable AND #Pump_Run_PB_Slew;
   IF #_w1 THEN #Pump_SP := 0.0; END_IF;
   #Pump_Run := #_w1;
   IF #_w1 THEN #Pump_Run_PB_Slew := FALSE; END_IF;
END_REGION
END_FUNCTION_BLOCK

FUNCTION_BLOCK "Door_Lock_Control"   // FB4, LAD
{ S7_Optimized_Access := 'TRUE' }
VERSION : 0.1
   VAR_INPUT
      Process_Complete : Bool;
      Rad_Lock : Bool;
      Safety_Key_Inserted : Bool;
      Door_Lock_Bypass : Bool;
   END_VAR
   VAR_OUTPUT
      Safety_Lock_Open : Bool;
   END_VAR
   VAR
      Safety_Lock_On : Bool;
      Edge_data_bit_1 : Bool;
      Edge_data_bit_2 : Bool;
      Door_Bypass_Alarm : Bool;
      Edge_data_bit_3 : Bool;
   END_VAR
   VAR_TEMP   // added for the SCL form of the ladder/FBD networks
      _w1 : Bool;
      _w2 : Bool;
   END_VAR
BEGIN

REGION Network 1
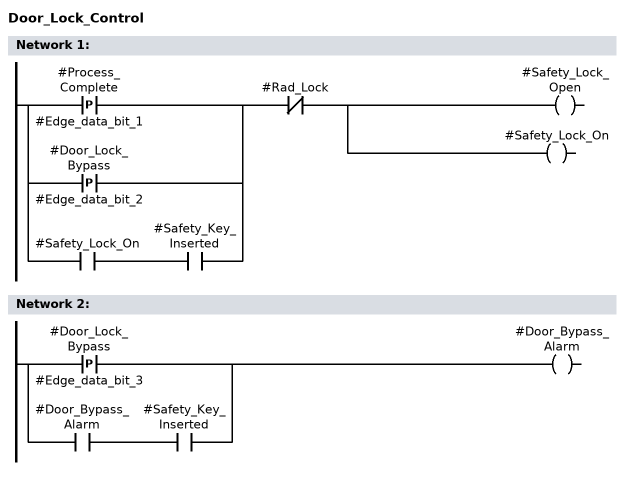
   RUNG wire#powerrail
      P_Contact(operand := #Process_Complete, bit := #Edge_data_bit_1)
      wire#w1
      I_Contact( #Rad_Lock )
      wire#w2
      Coil( #Safety_Lock_Open )
   END_RUNG
   RUNG wire#powerrail
      P_Contact(operand := #Door_Lock_Bypass, bit := #Edge_data_bit_2)
   END_RUNG wire#w1
   RUNG wire#powerrail
      Contact( #Safety_Lock_On )
      Contact( #Safety_Key_Inserted )
   END_RUNG wire#w1
   RUNG wire#w2
      Coil( #Safety_Lock_On )
   END_RUNG
   // the same network as SCL:
   #_w1 := #Process_Complete AND NOT #Edge_data_bit_1;   // rising edge of #Process_Complete
   #Edge_data_bit_1 := #Process_Complete;
   #_w2 := #Door_Lock_Bypass AND NOT #Edge_data_bit_2;   // rising edge of #Door_Lock_Bypass
   #Edge_data_bit_2 := #Door_Lock_Bypass;
   #Safety_Lock_Open := (#_w1 OR #_w2 OR (#Safety_Lock_On AND #Safety_Key_Inserted)) AND NOT #Rad_Lock;
   #Safety_Lock_On := #Safety_Lock_Open;
END_REGION

REGION Network 2
   RUNG wire#powerrail
      P_Contact(operand := #Door_Lock_Bypass, bit := #Edge_data_bit_3)
      wire#w1
      Coil( #Door_Bypass_Alarm )
   END_RUNG
   RUNG wire#powerrail
      Contact( #Door_Bypass_Alarm )
      Contact( #Safety_Key_Inserted )
   END_RUNG wire#w1
   // the same network as SCL:
   #_w1 := #Door_Lock_Bypass AND NOT #Edge_data_bit_3;   // rising edge of #Door_Lock_Bypass
   #Edge_data_bit_3 := #Door_Lock_Bypass;
   #Door_Bypass_Alarm := #_w1 OR (#Door_Bypass_Alarm AND #Safety_Key_Inserted);
END_REGION
END_FUNCTION_BLOCK

FUNCTION_BLOCK "Interlocks"   // FB5, LAD
{ S7_Optimized_Access := 'TRUE' }
VERSION : 0.1
// Logic used to set pump permissive to run, radiation interlocks, and estop interlocks.
   VAR_INPUT
      Vessel_Rad_Level : Real;
      Vessel_Rad_High_Alarm : Real;
      Pump_Rad_Level : Real;
      Pump_Rad_High_Alarm : Real;
      Estop1 : Bool;
      Estop2 : Bool;
      Safety_Relay_Trip : Bool;
      Safety_Lock_Engaged : Bool;
      Manual_Mode : Bool;
      Rad_Lock_Bypass : Bool;
      Process_Complete : Bool;
      Water_Supply_Interlock : Bool;
      UM_Container_Interlock : Bool;
      UM_Container_HH_Interlock : Bool;
      Buzzer_Reset : Bool;
   END_VAR
   VAR_OUTPUT
      Pump_Permisive : Bool;
   END_VAR
   VAR_IN_OUT
      Rad_Lock : Bool;
      Estop_Active : Bool;
      Level_Interlock : Bool;
   END_VAR
   VAR
      Vessel_Rad_Alarm : Bool;
      Pump_Rad_Alarm : Bool;
      Edge_Data_Bit : Bool;
   END_VAR
   VAR_TEMP   // added for the SCL form of the ladder/FBD networks
      _w1 : Bool;
   END_VAR
BEGIN

REGION Network 1
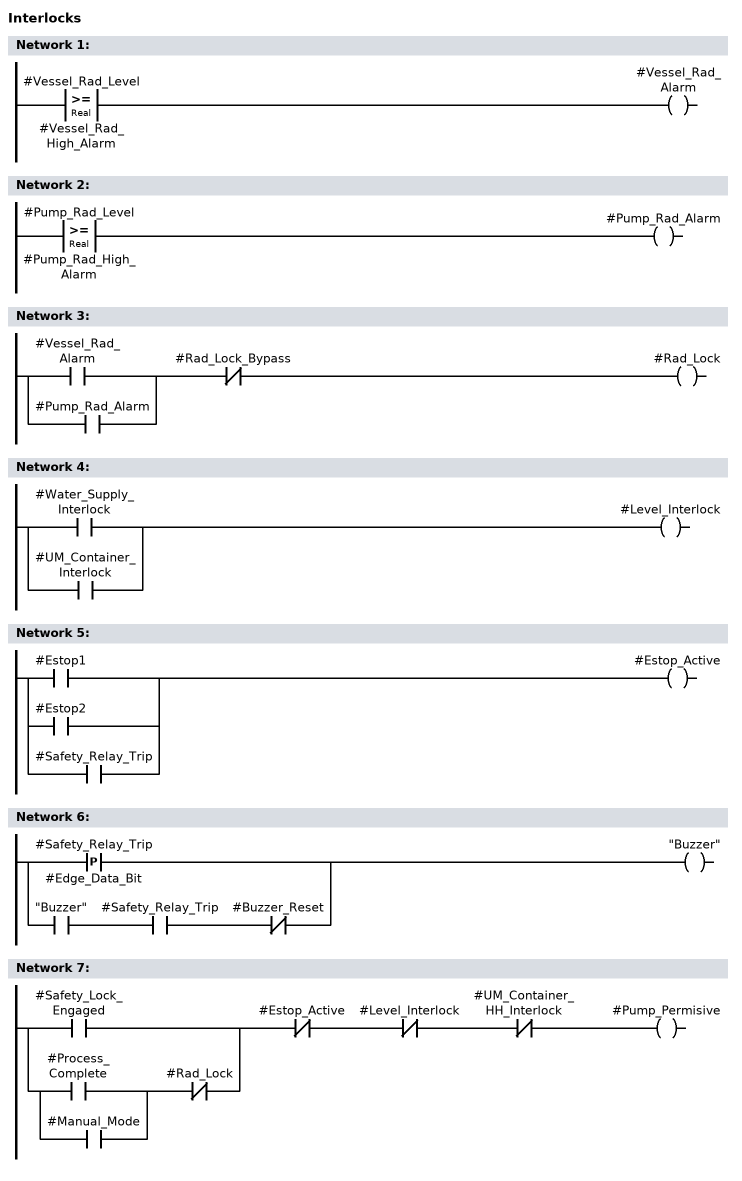
   RUNG wire#powerrail
      { S7_Templates := "SrcType := Real" } GE_Contact(in1 := #Vessel_Rad_Level, in2 := #Vessel_Rad_High_Alarm)
      Coil( #Vessel_Rad_Alarm )
   END_RUNG
   // the same network as SCL:
   #Vessel_Rad_Alarm := #Vessel_Rad_Level >= #Vessel_Rad_High_Alarm;
END_REGION

REGION Network 2
   RUNG wire#powerrail
      { S7_Templates := "SrcType := Real" } GE_Contact(in1 := #Pump_Rad_Level, in2 := #Pump_Rad_High_Alarm)
      Coil( #Pump_Rad_Alarm )
   END_RUNG
   // the same network as SCL:
   #Pump_Rad_Alarm := #Pump_Rad_Level >= #Pump_Rad_High_Alarm;
END_REGION

REGION Network 3
   RUNG wire#powerrail
      Contact( #Vessel_Rad_Alarm )
      wire#w1
      I_Contact( #Rad_Lock_Bypass )
      Coil( #Rad_Lock )
   END_RUNG
   RUNG wire#powerrail
      Contact( #Pump_Rad_Alarm )
   END_RUNG wire#w1
   // the same network as SCL:
   #Rad_Lock := (#Vessel_Rad_Alarm OR #Pump_Rad_Alarm) AND NOT #Rad_Lock_Bypass;
END_REGION

REGION Network 4
   RUNG wire#powerrail
      Contact( #Water_Supply_Interlock )
      wire#w1
      Coil( #Level_Interlock )
   END_RUNG
   RUNG wire#powerrail
      Contact( #UM_Container_Interlock )
   END_RUNG wire#w1
   // the same network as SCL:
   #Level_Interlock := #Water_Supply_Interlock OR #UM_Container_Interlock;
END_REGION

REGION Network 5
   RUNG wire#powerrail
      Contact( #Estop1 )
      wire#w1
      Coil( #Estop_Active )
   END_RUNG
   RUNG wire#powerrail
      Contact( #Estop2 )
   END_RUNG wire#w1
   RUNG wire#powerrail
      Contact( #Safety_Relay_Trip )
   END_RUNG wire#w1
   // the same network as SCL:
   #Estop_Active := #Estop1 OR #Estop2 OR #Safety_Relay_Trip;
END_REGION

REGION Network 6
   RUNG wire#powerrail
      P_Contact(operand := #Safety_Relay_Trip, bit := #Edge_Data_Bit)
      wire#w1
      Coil( "Buzzer" )
   END_RUNG
   RUNG wire#powerrail
      Contact( "Buzzer" )
      Contact( #Safety_Relay_Trip )
      I_Contact( #Buzzer_Reset )
   END_RUNG wire#w1
   // the same network as SCL:
   #_w1 := #Safety_Relay_Trip AND NOT #Edge_Data_Bit;   // rising edge of #Safety_Relay_Trip
   #Edge_Data_Bit := #Safety_Relay_Trip;
   "Buzzer" := #_w1 OR ("Buzzer" AND #Safety_Relay_Trip AND NOT #Buzzer_Reset);
END_REGION

REGION Network 7
   RUNG wire#powerrail
      Contact( #Safety_Lock_Engaged )
      wire#w1
      I_Contact( #Estop_Active )
      I_Contact( #Level_Interlock )
      I_Contact( #UM_Container_HH_Interlock )
      Coil( #Pump_Permisive )
   END_RUNG
   RUNG wire#powerrail
      Contact( #Process_Complete )
      wire#w2
      I_Contact( #Rad_Lock )
   END_RUNG wire#w1
   RUNG wire#powerrail
      Contact( #Manual_Mode )
   END_RUNG wire#w2
   // the same network as SCL:
   #Pump_Permisive := (#Safety_Lock_Engaged OR ((#Process_Complete OR #Manual_Mode) AND NOT #Rad_Lock)) AND NOT #Estop_Active AND NOT #Level_Interlock AND NOT #UM_Container_HH_Interlock;
END_REGION
END_FUNCTION_BLOCK

FUNCTION_BLOCK "Auto_Mode"   // FB6, SCL
{ S7_Optimized_Access := 'TRUE' }
VERSION : 0.1
   VAR_INPUT
      Pump_Remove_Full_Speed : Real;
      Ramp_Remove_Step : Int;
      Ramp_Remove_Time : Time;
      Pump_Drain_Full_Speed : Real;
      Ramp_Drain_Step : Int;
      Ramp_Drain_Time : Time;
      Pump_Rinse_Full_Speed : Real;
      Ramp_Rinse_Step : Int;
      Ramp_Rinse_Time : Time;
      Run_Drain_Time : Time;
      Run_Rinse_Time : Time;
      Run_Remove_Time : Time;
      Number_of_Rinses : Int;
      Abort_Stop : Bool;
      Use_RAD_CTRL : Bool;
      Pump_Cave_RAD_Level : Real;
      Rinse_To_RAD_Level : Real;
      Pump_Factor : Real;
      Pump_Stroke_Volume : Real;
   END_VAR
   VAR_OUTPUT
      Pump_Direction_FWD : Bool;
      Pump_Direction_REV : Bool;
      Valve_Direction : Bool;
      Pump_Run : Bool;
      Pump_Enable : Bool;
      Process_Complete : Bool;
      Pump_Speed : Real;
      Current_Rinse : Int;
      Current_Process_State : String;
   END_VAR
   VAR_IN_OUT
      Total_Flow_from_Supply : Real;
      Total_Flow_to_Waste : Real;
      Water_Container_Reset : Bool;
      Waste_Container_Reset : Bool;
      Run_State : Int;
   END_VAR
   VAR
      Total_Water_Supply_Update : Real;
      Convert_Water_Supply_Update : Real;
      Water_Update : Bool;
      Total_Waste_Drum_Update : Real;
      Convert_Waste_Drum_Update : Real;
      Waste_Drum_Update : Bool;
      Pump_to_UM_Full_Speed : Real;
      Ramp_UM_Step : Int;
      Ramp_UM_Time : Time;
      Run_UM_Time : Time;
      To_UM_State : String;
      "Step" : Int;
      Index : Int;
      Drain_Complete : Bool;
      Drain_Complete_Trig : Bool;
      Rinse_Complete : Bool;
      First_Pass_Complete : Bool;
      Rinse_Complete_Trig : Bool;
      Ready_Final_Drain : Bool;
      Delay_Time : Time := T#1s;
      At_RAD_Level : Bool;
      RAD_Complete_Rinses : Int;
      Current_Flow_to_Waste : Real;
      Current_Flow_from_Supply : Real;
      At_RAD_Level_Trig : Bool;
      Process_Complete_Trig : Bool;
      Waste_Container_Reset_Alarm : Bool;
      Water_Container_Reset_Alarm : Bool;
      Pump_Control_Instance_1 : "Pump_Control";
      R_TRIG_Instance : R_TRIG;
      Pump_Control_Instance_2 : "Pump_Control";
      R_TRIG_Instance_1 : R_TRIG;
      Pump_Control_Instance_3 : "Pump_Control";
      Delay_Timer_0_Instance : TON_TIME;
      R_TRIG_Instance_2 : R_TRIG;
      R_TRIG_Instance_3 : R_TRIG;
   END_VAR
   VAR CONSTANT
      INIT : Int := 1;
      RUN : Int := 10;
      STOP : Int := 20;
   END_VAR
BEGIN
   (*Function Block - Auto Mode: Control routine for automated Rinse/Drain Cycle.
   Called by: Automated Run (FB2)
   Calls: Pump CTRL (FB8) - 3 Instances (stored in this FB data instance)
   *)

   // Set CASE step as current run state
   #"Step" := #Run_State;

   CASE #"Step" OF
       #INIT:
           // Initialize variables
           #Waste_Container_Reset_Alarm := FALSE;
           #Water_Container_Reset_Alarm := FALSE;
           #First_Pass_Complete := FALSE;
           #Drain_Complete:=FALSE;
           #Process_Complete := FALSE;
           #Ready_Final_Drain := FALSE;
           #At_RAD_Level := FALSE;
           #Pump_Enable := FALSE;
           #Index := 0;
           #RAD_Complete_Rinses := 0;
           #Current_Process_State := 'INIT'; //For HMI

           // Look for trigger that PV is lower than the RAD CTRL SP (RAD control only)
           #R_TRIG_Instance_2(CLK := #At_RAD_Level,
                              Q => #At_RAD_Level_Trig);

           // Intialize both DRAIN state Pump CTRL instances

           #Pump_Control_Instance_1(Run_State:=#Run_State);
           #Pump_Control_Instance_2(Run_State:=#Run_State);

           #Pump_Control_Instance_3(Run_State := #Run_State);

           // Initialize pump and valve to waste
           #Pump_Direction_FWD := TRUE; // Forward
           #Pump_Direction_REV := FALSE;
           #Valve_Direction := FALSE; // to waste

       // CASE - Rinse process running    
       #RUN:
           #Pump_Enable := TRUE;

           // Currently not in final DRAIN step
           IF #Ready_Final_Drain = FALSE THEN

               IF NOT (#First_Pass_Complete) THEN
                   #To_UM_State := 'REMOVE';
                   #Pump_to_UM_Full_Speed := #Pump_Remove_Full_Speed;
                   #Ramp_UM_Step := #Ramp_Remove_Step;
                   #Ramp_UM_Time := #Ramp_Remove_Time;
                   #Run_UM_Time := #Run_Remove_Time;
               ELSE
                   #To_UM_State := 'DRAIN';
                   #Pump_to_UM_Full_Speed := #Pump_Drain_Full_Speed;
                   #Ramp_UM_Step := #Ramp_Drain_Step;
                   #Ramp_UM_Time := #Ramp_Drain_Time;
                   #Run_UM_Time := #Run_Drain_Time;
               END_IF;

                   //Remove residule fluid
                   #Current_Process_State := #To_UM_State; //For HMI
                   // Pump CTRL instance to pump to waste
                   #Pump_Control_Instance_1(Speed_SP_RPM := #Pump_to_UM_Full_Speed,
                                            Ramp_Steps := #Ramp_UM_Step,
                                            Ramp_Time := #Ramp_UM_Time,
                                            Steady_Run_Time := #Run_UM_Time,
                                            Run_State := #Run_State,
                                            Pump_Factor := #Pump_Factor,
                                            Pump_Stroke_Volume := #Pump_Stroke_Volume,
                                            Process_Complete => #Drain_Complete,
                                            Pump_Speed => #Pump_Speed,
                                            Pump_Run => #Pump_Run,
                                            Current_Total_flow => #Current_Flow_to_Waste);


                   // Look for trigger that Process State DRAIN is complete
                   #R_TRIG_Instance(CLK := #Drain_Complete,
                                    Q => #Drain_Complete_Trig);

                   // DRAIN state complete - initialize next pump instance (RINSE)
                   IF #Drain_Complete_Trig = TRUE THEN
                       #Total_Flow_to_Waste := #Total_Flow_to_Waste + #Current_Flow_to_Waste; // Totalilzer
                       #Run_State := #INIT;
                       #Pump_Control_Instance_2(Run_State := #Run_State);
                   END_IF;



               // Delay Start of Process State RINSE
               #Delay_Timer_0_Instance(IN := #Drain_Complete,
                                       PT := #Delay_Time);


               // Run RINSE state when delay timer complete    
           IF #Drain_Complete = TRUE AND #Delay_Timer_0_Instance.Q = TRUE THEN
                   // Run RINSE cycle
               #First_Pass_Complete := TRUE;

                   #Pump_Direction_FWD := FALSE;
                   #Pump_Direction_REV := TRUE; // Reverse
                   #Valve_Direction := TRUE; // From water supply 
                   #Run_State := #RUN;

                   #Current_Process_State := 'RINSE'; //For HMI
                   // Pump CTRL instance to RINSE - water from supply to vessel
                   #Pump_Control_Instance_2(Speed_SP_RPM := #Pump_Rinse_Full_Speed,
                                           Ramp_Steps := #Ramp_Rinse_Step,
                                           Ramp_Time := #Ramp_Rinse_Time,
                                           Steady_Run_Time := #Run_Rinse_Time,
                                           Run_State := #Run_State,
                                           Pump_Factor:=#Pump_Factor,
                                           Pump_Stroke_Volume:=#Pump_Stroke_Volume,
                                           Process_Complete => #Rinse_Complete,
                                           Pump_Speed => #Pump_Speed,
                                           Pump_Run => #Pump_Run,
                                           Current_Total_flow=> #Current_Flow_from_Supply);
               END_IF;

               // Look for trigger that Process State RINSE is complete
               #R_TRIG_Instance_1(CLK := #Rinse_Complete,
                                  Q => #Rinse_Complete_Trig);

               // RINSE state complete - initialize next pump CTRL instance (WASTE)
               IF #Rinse_Complete_Trig = TRUE THEN

                   #Total_Flow_from_Supply := #Total_Flow_from_Supply + #Current_Flow_from_Supply; // Totalizer
                   #Index := #Index + 1; // Count last rinse cycle for HMI
                   #Run_State := #INIT;
                   #Pump_Control_Instance_1(Run_State := #Run_State);
               END_IF;

               // Run DRAIN state
               IF #Rinse_Complete = TRUE THEN
                  // #First_Pass_Complete := TRUE;
                   #Pump_Direction_FWD := TRUE; // Forward
                   #Pump_Direction_REV := FALSE;
                   #Valve_Direction := FALSE; // To waste

                   // RAD CTRL Logic - if selected will contine to rinse until RAD level drops below SP
                   IF #Use_RAD_CTRL = TRUE THEN
                       IF #Pump_Cave_RAD_Level < #Rinse_To_RAD_Level THEN
                           #At_RAD_Level := TRUE;
                       END_IF;

                       // Look for trigger that RAD level has dropped below SP
                       #R_TRIG_Instance_2(CLK := #At_RAD_Level,
                                          Q => #At_RAD_Level_Trig);

                       // RAD CTRL counters for HMI
                       IF #At_RAD_Level_Trig = TRUE THEN
                           #RAD_Complete_Rinses := #Number_of_Rinses + #Index;
                       END_IF;

                       // If RAD level drops below SP and final rinses complete - run final DRAIN state
                       IF (#Index = #RAD_Complete_Rinses) AND (#At_RAD_Level = TRUE) THEN
                           #Ready_Final_Drain := TRUE;
                       END_IF;

                   ELSE
                       // Not using RAD CTRl - check to see if completed all rinses
                       IF #Index = #Number_of_Rinses THEN
                           #Ready_Final_Drain := TRUE; // Run final DRAIN state
                       END_IF;

                   END_IF; // RAD CTRL statement
               END_IF; // Rinse complete statement
           END_IF; // Ready for final drain statement

           // Ready to run final DRAIN cycle to remove remaining liquid from vessel
           IF #Ready_Final_Drain = TRUE THEN
               //Run DRAIN Cycle
               #Pump_Direction_FWD := TRUE; // Forward
               #Pump_Direction_REV := FALSE;
               #Valve_Direction := FALSE; // To Waste
               #Run_State := #RUN;
               #Current_Process_State := 'DRAIN'; //For HMI

               // Pump CTRL instance to DRAIN (final)
               #Pump_Control_Instance_3(Speed_SP_RPM := #Pump_Drain_Full_Speed,
                                       Ramp_Steps := #Ramp_Drain_Step,
                                       Ramp_Time := #Ramp_Drain_Time,
                                       Steady_Run_Time := #Run_Drain_Time,
                                       Run_State := #Run_State,
                                       Pump_Factor:=#Pump_Factor,
                                       Pump_Stroke_Volume:=#Pump_Stroke_Volume,
                                       Process_Complete => #Process_Complete,
                                       Pump_Speed => #Pump_Speed,
                                       Pump_Run => #Pump_Run,
                                       Current_Total_flow=> #Current_Flow_to_Waste);
               #R_TRIG_Instance_3(CLK:=#Process_Complete,
                                  Q=>#Process_Complete_Trig);

               IF #Process_Complete_Trig = TRUE THEN
                   #Total_Flow_to_Waste := #Total_Flow_to_Waste + #Current_Flow_to_Waste; // Totalilzer
               END_IF;

           END_IF; // Final Drain statement

           #Current_Rinse := #Index; //Pass through for HMI

       // CASE - stop process    
       #STOP:
           #Pump_Speed := 0.0;

          #Pump_Run := TRUE;


           #Pump_Direction_FWD := TRUE; // Set direction forward (failsafe)
           #Pump_Direction_REV := FALSE;
           #Valve_Direction := FALSE; // Set vavle to waste (failsafe)
           IF #Abort_Stop = TRUE THEN // For HMI
               #Current_Process_State := 'ABORT';
           ELSE
               #Current_Process_State := 'COMPLETE';
           END_IF;

           IF #Water_Container_Reset = TRUE THEN
               #Total_Flow_from_Supply := 0.0;
               #Water_Container_Reset_Alarm := TRUE;
               #Water_Container_Reset := FALSE;
           END_IF;

           IF #Water_Update = TRUE THEN
               #Convert_Water_Supply_Update := #Total_Water_Supply_Update * 10000;
               #Total_Flow_from_Supply := #Total_Flow_from_Supply + #Convert_Water_Supply_Update;
               #Total_Water_Supply_Update := 0.0;
               #Water_Update := FALSE;
           END_IF;

           IF #Waste_Container_Reset = TRUE THEN
               #Total_Flow_to_Waste := 0.0;
               #Waste_Container_Reset_Alarm := TRUE;
               #Waste_Container_Reset := FALSE;
           END_IF;

           IF #Waste_Drum_Update = TRUE THEN
               #Convert_Waste_Drum_Update := #Total_Waste_Drum_Update * 10000;
               #Total_Flow_to_Waste := #Total_Flow_to_Waste + #Convert_Waste_Drum_Update;
               #Total_Waste_Drum_Update := 0.0;
               #Waste_Drum_Update := FALSE;
           END_IF;


   END_CASE;
END_FUNCTION_BLOCK

FUNCTION_BLOCK "Discrete_Alarm_Source"   // FB7, SCL
{ S7_Optimized_Access := 'TRUE' }
VERSION : 0.1
   VAR
      Alarm_Integer_1 : Int;
      Alarm_Integer_2 : Int;
   END_VAR
BEGIN



   "Convert_16bits_to_Integer"(bit0:="Estop1_PB_Active",
                               bit1:="Estop2_PB_Active",
                               bit2:="Safety_Relay_Trip",
                               bit3:="S1_General_Setup".Rad_Lock,
                               bit4:="S2_General_Setup".Rad_Lock,
                               bit5:="S1_General_Setup".Rad_Lock_Bypass,
                               bit6:="S2_General_Setup".Rad_Lock_Bypass,
                               bit7:="S1_ Door_Lock_Control_DB".Door_Bypass_Alarm,
                               bit8:="S2_Door_Lock_Control_DB".Door_Bypass_Alarm,
                               bit9:="S1_Automated_Run_DB".Auto_Mode_Instance.Waste_Container_Reset_Alarm,
                               bit10:="S1_Automated_Run_DB".Auto_Mode_Instance.Water_Container_Reset_Alarm,
                               bit11:="S2_Automated_Run_DB".Auto_Mode_Instance.Water_Container_Reset_Alarm,
                               bit12:="S1_General_Setup".Water_Supply_Interlock,
                               bit13:="S2_General_Setup".Water_Supply_Interlock,
                               bit14:="Setup_Data".Waste_Container_Interlock,
                               bit15:=FALSE,
                               Value=>#Alarm_Integer_1);

   "Convert_16bits_to_Integer"(bit0 := "S1_General_Setup".Pump_Error_Bit,
                               bit1 := "S2_General_Setup".Pump_Error_Bit,
                               bit2 := "UM_HI_Level_SW",
                               bit3 := "S1_Automated_Run_DB".Pump_Fail_Alarm,
                               bit4 := "S2_Automated_Run_DB".Pump_Fail_Alarm,
                               bit5 := FALSE,
                               bit6 := FALSE,
                               bit7 := FALSE,
                               bit8 := FALSE,
                               bit9 := FALSE,
                               bit10 := FALSE,
                               bit11 := FALSE,
                               bit12 := FALSE,
                               bit13 := FALSE,
                               bit14 := FALSE,
                               bit15 := FALSE,
                               Value => #Alarm_Integer_2);
END_FUNCTION_BLOCK

FUNCTION_BLOCK "Integration"   // FB10, SCL
{ S7_Optimized_Access := 'TRUE' }
VERSION : 0.1
   VAR_INPUT
      in : DInt;
      enable : Bool;
      reset : Bool;
   END_VAR
   VAR_OUTPUT
      out : LReal;
      error : Bool;
   END_VAR
   VAR
      actualTime : DTL;
      lastTime : DTL;
      statIn : LReal;
      lastIn : LReal;
      integral : LReal;
   END_VAR
   VAR_TEMP
      deltaTimeT : Time;
      deltaTimeDI : DInt;
      deltaTime : LReal;
      rv1 : Int;
      tempAux : LReal;
   END_VAR
BEGIN
   //Der Eingangswert am Eingang "in" wird mit Hilfe des FB "Integration" integriert.
   //Am Parameter "out" des FBs erfolgt die Ausgabe des Integralwertes und wird remanent gehalten.
   // - "reset" setzt den Ausgabewert des Integrationsbausteins zurück.
   // - "enable" startet die Integralberechnung und ist remanent zu wählen, wenn die Integration nach einem Spannungsausfall fortgesetzt werden soll.
   // - das Ausgangsbit "error" signalisiert die fehlende Aktivierung oder Beschaltung des Systemmerkerbyte. Ist das "Error"-Bit nur für einen Zyklus aktiv, trat eine Spannungswiederkehr während der Integration auf.
   //*******************************************************************************************************************************************************************************************************************
   //The input value "in" will be integrated by the FB "Integration".
   //The output value of the "Integration" is the parameter "out" and is retentive and holds the integrated value.
   // - "reset" resets the integrated output value "out".
   // - "enable" starts the integral calculation and must be retentive if the integration should continue after a power failure.
   // - the output bit "error" signals that the system memory byte is disabled or not connected (when glowing). Is active for one cycle only, it signals a power up while integration.

    IF #reset = true THEN
        #out := 0.0;
        #lastIn := 0.0;
        #integral := 0.0;
        RETURN;
    END_IF;

   #tempAux:= NORM_X(MIN:=0, VALUE:=#in, MAX:=27648);
   #statIn:= SCALE_X(MIN:=0.0, VALUE:=#tempAux, MAX:=10.0);

   #rv1:= RD_SYS_T(OUT=>#actualTime);

   #deltaTimeT:= T_DIFF(IN1:=#actualTime, IN2:=#lastTime);
   #deltaTimeDI:= T_CONV(#deltaTimeT);

   #deltaTime:= DINT_TO_LREAL(#deltaTimeDI);
   #deltaTime := #deltaTime / 1000.0;
   #lastTime := #actualTime;

   IF NOT #enable = true THEN
       #lastIn := 0.0;
       RETURN;
   END_IF;

   #statIn := #statIn + #lastIn;
   #statIn := #statIn / 2.0;
   #statIn := #statIn * #deltaTime;
   #integral := #integral + #statIn;
   #out:= #integral;

   #lastIn := #statIn;
END_FUNCTION_BLOCK

FUNCTION_BLOCK "Motor_Control"   // FB12, SCL
{ S7_Optimized_Access := 'TRUE' }
VERSION : 0.1
   VAR_INPUT
      Pump_Run_Enable : Bool;
      HW_Address_I : Hw_Io;
      HW_Address_O : Hw_Io;
   END_VAR
   VAR_OUTPUT
      Pump_Vel_Feedback : Real;
      Pump_En_Feedback : DInt;
      Pump_Error_Code : UInt;
      Pump_Error_Bit : Bool;
   END_VAR
   VAR_IN_OUT
      Settings : "UDT_MDrive_Settings";
      Token : "UDT_MDrive_Data";
   END_VAR
   VAR
      Pump : "M_Drive";
   END_VAR
BEGIN



   #Pump(Enable:= #Pump_Run_Enable,
         HW_Address_I:=#HW_Address_I,
         HW_Address_O:=#HW_Address_O,
         Settings:=#Settings,
         Token:=#Token);



   #Pump_Vel_Feedback := #Pump.Drive_PIW.V;
   #Pump_En_Feedback := #Pump.Drive_PIW.C2;

   #Pump_Error_Code := #Pump.Drive_PIW.Error;

   IF #Pump_Error_Code > 0 THEN
       #Pump_Error_Bit := TRUE;
   ELSE
       #Pump_Error_Bit := FALSE;
   END_IF;
END_FUNCTION_BLOCK

FUNCTION_BLOCK "Pump_Control"   // FB13, SCL
{ S7_Optimized_Access := 'TRUE' }
VERSION : 0.1
   VAR_INPUT
      Speed_SP_RPM : Real;
      Ramp_Steps : Int;
      Ramp_Time : Time;
      Steady_Run_Time : Time;
      Run_State : Int;
      Hold_Run_Timer : Bool;
      Pump_Factor : Real;
      Pump_Stroke_Volume : Real;
   END_VAR
   VAR_OUTPUT
      Process_Complete : Bool;
      Pump_Speed : Real;
      Pump_Run : Bool;
      Current_Total_flow : Real;
   END_VAR
   VAR
      Ramp_Up_Complete : Bool;
      Ramp_Down_Complete : Bool;
      "Step" : Int;
      Speed_SP : Real;
      Ramp_Setpoint : Real;
      Ramp_Speed : Real;
      Pump_Lower_Limit : Real := 0.0;
      Speed_Lower_Limit : Real := 50.0;
      Enable_Integration : Bool;
      Reset_Integration : Bool;
      Current_flow_rate : DInt;
      RampUp_Timer_0_Instance : TOF_TIME;
      Run_Timer_0_Instance_1 : TON_TIME;
      R_TRIG_Instance : R_TRIG;
      New_Ramp : Bool;
      Curr_Ramp_Step : Int;
      RampDown_Timer_0_Instance : TOF_TIME;
      Integration_Instance : "Integration";
      R_TRIG_Instance_1 : R_TRIG;
      R_TRIG_Instance_2 : R_TRIG;
      R_TRIG_Instance_3 : R_TRIG;
      R_TRIG_Instance_4 : R_TRIG;
   END_VAR
   VAR_TEMP
      Setpoint_change : Bool;
   END_VAR
   VAR CONSTANT
      INIT : Int := 1;
      RUN : Int := 10;
      STOP : Int := 20;
   END_VAR
BEGIN

   #"Step" := #Run_State;



   CASE #"Step" OF
       #INIT:
           #Pump_Run := FALSE;
           #Ramp_Up_Complete := FALSE;
           #Ramp_Down_Complete := FALSE;
           #Process_Complete := FALSE;
           #Reset_Integration := TRUE;

           // Ramp up Init
           #Curr_Ramp_Step := 0;
           #Ramp_Setpoint := 0.0;
           #Ramp_Speed := 0.0;
           #Pump_Speed := #Ramp_Speed;


       #RUN:
           #Pump_Run := FALSE;
           #Enable_Integration := TRUE;
           #Reset_Integration := FALSE;


           "Pump_RPM_Conversion"(Speed_SP_RPM:=#Speed_SP_RPM,
                                 Speed_SP_Counts=>#Speed_SP);

           // Ramp Up
           IF NOT (#Ramp_Up_Complete) THEN
               #Ramp_Setpoint := #Speed_SP / #Ramp_Steps;

               IF NOT (#RampUp_Timer_0_Instance.Q) AND NOT (#Ramp_Up_Complete) THEN
                   #Ramp_Speed := #Ramp_Setpoint + #Ramp_Speed;
                   IF #Ramp_Speed > #Speed_SP THEN
                       #Ramp_Speed := #Speed_SP;
                   END_IF;
                   #Pump_Speed := #Ramp_Speed;
                   #Setpoint_change := TRUE;
                   #Curr_Ramp_Step := #Curr_Ramp_Step + 1;

                   #Pump_Run := TRUE;
               ELSE
                   #Setpoint_change := FALSE;
                   #Pump_Run := FALSE;
               END_IF;

               #RampUp_Timer_0_Instance(IN := #Setpoint_change,
                                        PT := #Ramp_Time);

           IF #Curr_Ramp_Step > #Ramp_Steps THEN
               #Ramp_Up_Complete := TRUE;
               #Pump_Run := TRUE;
           ELSE
               #Ramp_Up_Complete := FALSE;
           END_IF;

       END_IF;


       // Run Steady state
       IF #Hold_Run_Timer = TRUE THEN
          RETURN;
      END_IF;
               #Run_Timer_0_Instance_1(IN := #Ramp_Up_Complete,
                                       PT := #Steady_Run_Time);

               #R_TRIG_Instance(CLK := #Run_Timer_0_Instance_1.Q,
                                Q => #New_Ramp);

               IF #New_Ramp = TRUE THEN
                   #Pump_Speed := 0.0;
                   #Pump_Run := TRUE;
                   #Process_Complete := TRUE;

               END_IF;


           #STOP:

          #Enable_Integration := FALSE;


   END_CASE;


   // pump flow
   #Current_flow_rate := #Pump_Factor * #Pump_Stroke_Volume * #Pump_Speed;
   #Integration_Instance(in := #Current_flow_rate,
                         enable := #Enable_Integration,
                         reset := #Reset_Integration,
                         out => #Current_Total_flow);
END_FUNCTION_BLOCK

FUNCTION_BLOCK "Pump_HMI"   // FB14, LAD
{ S7_Optimized_Access := 'TRUE' }
VERSION : 0.1
   VAR_INPUT
      Pump_Vel_Feedback : Real;
      Pump_En_Feedback : DInt;
   END_VAR
   VAR_OUTPUT
      Pump_Run_En : Bool;
      Feedback_RPM : Real;
   END_VAR
   VAR_IN_OUT
      Pump_Run : Bool;
   END_VAR
   VAR
      Pump_Feedback_Abs : Real;
      Pump_FWD : Bool;
      Pump_REV : Bool;
      Pump_En_Hold : DInt;
      Pump_En_Diff : DInt;
      Pump_En_Abs : DInt;
   END_VAR
   VAR CONSTANT
      Pump_En_Required_Change : DInt := 5;
   END_VAR
BEGIN

REGION Network 1
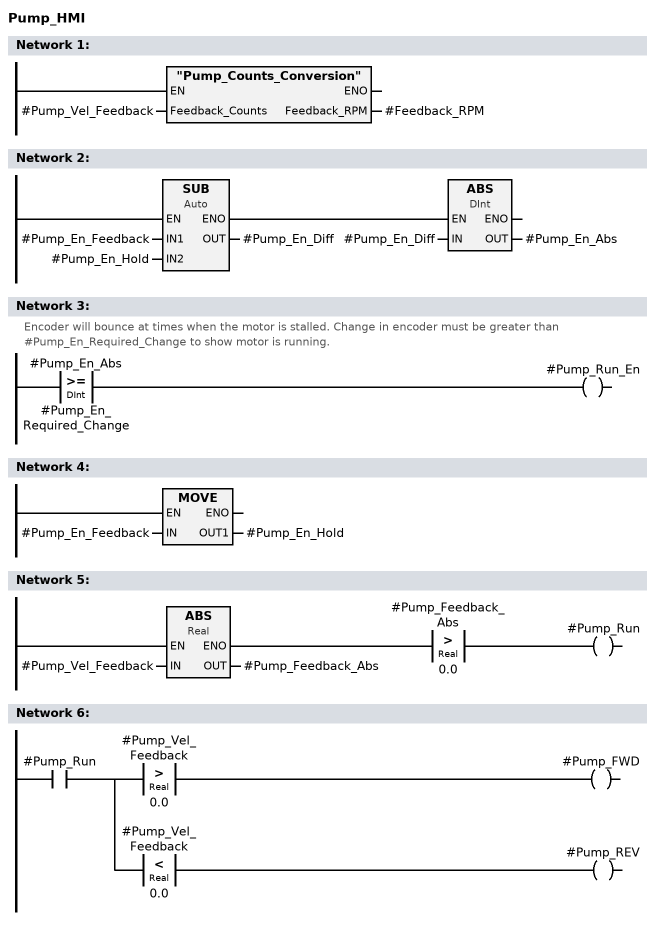
   RUNG wire#powerrail
      "Pump_Counts_Conversion"(Feedback_Counts := #Pump_Vel_Feedback, Feedback_RPM => #Feedback_RPM)
   END_RUNG
   // the same network as SCL:
   "Pump_Counts_Conversion"(Feedback_Counts := #Pump_Vel_Feedback, Feedback_RPM => #Feedback_RPM);
END_REGION

REGION Network 2
   RUNG wire#powerrail
      Sub(in1 := #Pump_En_Feedback, in2 := #Pump_En_Hold, out => #Pump_En_Diff)
      { S7_Templates := "SrcType := DInt" } Abs(in := #Pump_En_Diff, out => #Pump_En_Abs)
   END_RUNG
   // the same network as SCL:
   #Pump_En_Diff := #Pump_En_Feedback - #Pump_En_Hold;
   #Pump_En_Abs := ABS(#Pump_En_Diff);
END_REGION

REGION Network 3
   // Encoder will bounce at times when the motor is stalled. Change in encoder must be greater than #Pump_En_Required_Change to show motor is running.
   RUNG wire#powerrail
      { S7_Templates := "SrcType := DInt" } GE_Contact(in1 := #Pump_En_Abs, in2 := #Pump_En_Required_Change)
      Coil( #Pump_Run_En )
   END_RUNG
   // the same network as SCL:
   #Pump_Run_En := #Pump_En_Abs >= #Pump_En_Required_Change;
END_REGION

REGION Network 4
   RUNG wire#powerrail
      Move(in := #Pump_En_Feedback, out1 => #Pump_En_Hold)
   END_RUNG
   // the same network as SCL:
   #Pump_En_Hold := #Pump_En_Feedback;
END_REGION

REGION Network 5
   RUNG wire#powerrail
      { S7_Templates := "SrcType := Real" } Abs(in := #Pump_Vel_Feedback, out => #Pump_Feedback_Abs)
      { S7_Templates := "SrcType := Real" } GT_Contact(in1 := #Pump_Feedback_Abs, in2 := 0.0)
      Coil( #Pump_Run )
   END_RUNG
   // the same network as SCL:
   #Pump_Feedback_Abs := ABS(#Pump_Vel_Feedback);
   #Pump_Run := #Pump_Feedback_Abs > 0.0;
END_REGION

REGION Network 6
   RUNG wire#powerrail
      Contact( #Pump_Run )
      wire#w1
      { S7_Templates := "SrcType := Real" } GT_Contact(in1 := #Pump_Vel_Feedback, in2 := 0.0)
      Coil( #Pump_FWD )
   END_RUNG
   RUNG wire#w1
      { S7_Templates := "SrcType := Real" } LT_Contact(in1 := #Pump_Vel_Feedback, in2 := 0.0)
      Coil( #Pump_REV )
   END_RUNG
   // the same network as SCL:
   #Pump_FWD := #Pump_Run AND (#Pump_Vel_Feedback > 0.0);
   #Pump_REV := #Pump_Run AND (#Pump_Vel_Feedback < 0.0);
END_REGION
END_FUNCTION_BLOCK

FUNCTION_BLOCK "M_Drive"   // FB86, SCL
{ S7_Optimized_Access := 'FALSE' }
VERSION : 0.1
   VAR_INPUT
      Enable : Bool := False;
      HW_Address_I : Hw_Io;
      HW_Address_O : Hw_Io;
   END_VAR
   VAR_IN_OUT
      Token : "UDT_MDrive_Data";
      Settings : "UDT_MDrive_Settings";
   END_VAR
   VAR
      Drive_PIW : "UDT_MDrive_PIW";
      Drive_PQW : "UDT_MDrive_PQW";
      PQW_Data AT Drive_PQW : Array[0..63] of Word;
      "PQW_Data 1" : Bool;
      RetVal_WR : Int;
      RetVal_RD : Int;
      Tof_DriveMoving : TOF_TIME;
      Ton_ResetTrigger : TON_TIME;
      PIW_Inputs_Array : Array[0..7] of Bool;
      PIW_Inputs AT PIW_Inputs_Array : USInt;
      HMI_Data : "UDT_HMI_MDrive";
      Ton_ResetTrigger_All : TON_TIME;
      ton_start : TON_TIME;
      Ton_stop : TON_TIME;
      RT_ResetTrigger : R_TRIG;
      RT_ResetTriggerAll : R_TRIG;
   END_VAR
   VAR_TEMP
      L_Slew : DInt;
      L_S : DInt;
   END_VAR
   VAR CONSTANT
      Deviation : DInt := 5;
   END_VAR
   // Drive_PQW.R9_R10.Reg9 := False;
   // Drive_PQW.R9_R10.Bit1 := False;
   // Drive_PQW.R9_R10.Bit2 := False;
   // Drive_PQW.R9_R10.Bit3 := False;
   // Drive_PQW.R9_R10.Bit4 := False;
   // Drive_PQW.R9_R10.Bit5 := False;
   // Drive_PQW.R9_R10.Bit6 := False;
   // Drive_PQW.R9_R10.Bit7 := False;
   // Drive_PQW.R9_R10.Reg10 := False;
   // Drive_PQW.R9_R10.Bit8 := False;
   // Drive_PQW.R9_R10.Bit9 := False;
   // Drive_PQW.R9_R10.Bit10 := False;
   // Drive_PQW.R9_R10.Bit11 := False;
   // Drive_PQW.R9_R10.Bit12 := False;
   // Drive_PQW.R9_R10.Bit13 := False;
   // Drive_PQW.R9_R10.Bit14 := False;
   // Drive_PQW.R11.Reg11 := False;
   // Drive_PQW.R11.Bit1 := False;
   // Drive_PQW.R11.Bit2 := False;
   // Drive_PQW.R11.Bit3 := False;
   // Drive_PQW.R11.Bit4 := False;
   // Drive_PQW.R11.Bit5 := False;
   // Drive_PQW.R11.Bit6 := False;
   // Drive_PQW.R11.Bit7 := False;
   // Drive_PQW.R1_R38.Dummy_Bit0 := False;
   // Drive_PQW.R1_R38.Dummy_Bit1 := False;
   // Drive_PQW.R1_R38.Dummy_Bit2 := False;
   // Drive_PQW.R1_R38.Dummy_Bit3 := False;
   // Drive_PQW.R1_R38.Dummy_Bit4 := False;
   // Drive_PQW.R1_R38.Dummy_Bit5 := False;
   // Drive_PQW.R1_R38.Dummy_Bit6 := False;
   // Drive_PQW.R1_R38.Dummy_Bit7 := False;
   // Drive_PQW.R1_R38.Reg1 := False;
   // Drive_PQW.R1_R38.Reg2 := False;
   // Drive_PQW.R1_R38.Reg3 := False;
   // Drive_PQW.R1_R38.Reg4 := False;
   // Drive_PQW.R1_R38.Reg5 := False;
   // Drive_PQW.R1_R38.Reg6 := False;
   // Drive_PQW.R1_R38.Reg7 := False;
   // Drive_PQW.R1_R38.Reg8 := False;
   // Drive_PQW.R1_R38.Reg9 := False;
   // Drive_PQW.R1_R38.Reg10 := False;
   // Drive_PQW.R1_R38.Reg11 := False;
   // Drive_PQW.R1_R38.Reg12 := False;
   // Drive_PQW.R1_R38.Reg13 := False;
   // Drive_PQW.R1_R38.Reg14 := False;
   // Drive_PQW.R1_R38.Reg15 := False;
   // Drive_PQW.R1_R38.Reg16 := False;
   // Drive_PQW.R1_R38.Reg17 := False;
   // Drive_PQW.R1_R38.Reg18 := False;
   // Drive_PQW.R1_R38.Reg19 := False;
   // Drive_PQW.R1_R38.Reg20 := False;
   // Drive_PQW.R1_R38.Reg21 := False;
   // Drive_PQW.R1_R38.Reg22 := False;
   // Drive_PQW.R1_R38.Reg23 := False;
   // Drive_PQW.R1_R38.Reg24 := False;
   // Drive_PQW.R1_R38.Reg25 := False;
   // Drive_PQW.R1_R38.Reg26 := False;
   // Drive_PQW.R1_R38.Reg27 := False;
   // Drive_PQW.R1_R38.Reg28 := False;
   // Drive_PQW.R1_R38.Reg32 := False;
   // Drive_PQW.R1_R38.Reg33 := False;
   // Drive_PQW.R1_R38.Reg38 := False;
   // Drive_PQW.R1_R38.Dummy_Bit8 := False;
   // Drive_PQW.R1_R38.Dummy_Bit9 := False;
   // Drive_PQW.R1_R38.Dummy_Bit10 := False;
   // Drive_PQW.R1_R38.Dummy_Bit11 := False;
   // Drive_PQW.R1_R38.Dummy_Bit12 := False;
   // Drive_PQW.R1_R38.Dummy_Bit13 := False;
   // Drive_PQW.R1_R38.Dummy_Bit14 := False;
   // Drive_PQW.R1_R38.Dummy_Bit15 := False;
   // Drive_PQW.R1_R38.Dummy_Bit16 := False;
   // Tof_DriveMoving.IN := False;
   // Tof_DriveMoving.Q := False;
   // Ton_ResetTrigger.IN := False;
   // Ton_ResetTrigger.Q := False;
   // PIW_Inputs_Array[0] := False;
   // PIW_Inputs_Array[1] := False;
   // PIW_Inputs_Array[2] := False;
   // PIW_Inputs_Array[3] := False;
   // PIW_Inputs_Array[4] := False;
   // PIW_Inputs_Array[5] := False;
   // PIW_Inputs_Array[6] := False;
   // PIW_Inputs_Array[7] := False;
   // HMI_Data.Slew.Fwd := False;
   // HMI_Data.Slew.Rev := False;
   // HMI_Data.State.IsMoving := False;
   // HMI_Data.State.IsHomed := False;
   // HMI_Data.State.OnPosition := False;
   // Ton_ResetTrigger_All.IN := False;
   // Ton_ResetTrigger_All.Q := False;
   // ton_start.IN := False;
   // ton_start.Q := False;
   // Ton_stop.IN := False;
   // Ton_stop.Q := False;
BEGIN


   IF NOT #Enable THEN
       #Token.CMD_Trigger.Slew := False;
   END_IF;

   IF #Token.CMD_Trigger.Slew THEN // register 11
       //trigger needed...  +/- 2.000.000 

       IF #Token.Slew.Speed = 0 THEN
           #Token.Slew.Fwd := False;
           #Token.Slew.Rev := False;
       END_IF;

      #L_Slew := #Token.Slew.Speed;

       IF #Token.Slew.Fwd THEN
           #Drive_PQW.Slew := #L_Slew;
       ELSIF #Token.Slew.Rev THEN
           #Drive_PQW.Slew := - #L_Slew;
       ELSE
           #Drive_PQW.Slew := 0;
       END_IF;

       #Drive_PQW.R11.Reg11 := True;

   END_IF;

   #Drive_PQW.DriveEnable := 1;

   #Ton_ResetTrigger(IN := #Token.CMD_Busy,
                     PT := T#100ms);

   #Ton_ResetTrigger_All(IN := #Ton_ResetTrigger.Q,
                         PT := T#100ms);

   #RT_ResetTrigger(CLK := #Ton_ResetTrigger.Q);

   IF #PQW_Data[36].%B1 > 0 THEN
       #Token.CMD_Busy := True;
   ELSIF #Ton_ResetTrigger_All.Q THEN
       #Token.CMD_Busy := False;
   END_IF;


   IF #Ton_ResetTrigger.Q THEN
       #PQW_Data[36].%B1 := 16#0;
       #Token.CMD_Trigger.Slew := False;
   END_IF;

   #RetVal_WR := DPWR_DAT(LADDR := #HW_Address_O, RECORD := #Drive_PQW);

   #RetVal_RD := DPRD_DAT(LADDR := #HW_Address_I, RECORD => #Drive_PIW);

   #Tof_DriveMoving(IN := #Drive_PIW.MV > 0,
                    PT := T#50ms,
                    Q => #Token.State.IsMoving);

   #PIW_Inputs := #Drive_PIW.Inputs;
   #Token.Inputs := #PIW_Inputs_Array;

   IF #Token.Reset THEN
       #Drive_PQW.SetError := 0;
       #Drive_PQW.R1_R38.Reg15 := True;
   END_IF;
END_FUNCTION_BLOCK

FUNCTION "Pump_Counts_Conversion" : Void   // FC1, SCL
{ S7_Optimized_Access := 'TRUE' }
VERSION : 0.1
   VAR_INPUT
      Feedback_Counts : Real;
   END_VAR
   VAR_OUTPUT
      Feedback_RPM : Real;
   END_VAR
BEGIN

   #Feedback_RPM := #Feedback_Counts / 932;
END_FUNCTION

FUNCTION "UM_Vault_Calc" : Void   // FC2, SCL
{ S7_Optimized_Access := 'TRUE' }
VERSION : 0.1
   VAR_INPUT
      Total_Waste_from_Station1 : Real;
      Total_Waste_from_Station2 : Real;
      "Waste_Drum-Volume" : Real;
      Waste_Container_Alarm_SP : Real;
      Waste_Container_Interlock_Level : Real;
      Waste_Rad_Level : Real;
      "Waste_Rad_High-Alarm" : Real;
   END_VAR
   VAR_OUTPUT
      Total_Waste_Volume : Real;
      Total_Waste_Volume_Percent : Real;
      Waste_Container_Alarm_Level : Int;
      Waste_Container_Interlock : Bool;
      Waste_Rad_Alarm : Bool;
      Alarm_Green : Bool;
      Alarm_Red : Bool;
   END_VAR
BEGIN


   #Total_Waste_Volume := (#Total_Waste_from_Station1 + #Total_Waste_from_Station2) / 10000;
   #Total_Waste_Volume_Percent := (#Total_Waste_Volume / #"Waste_Drum-Volume" ) * 100;

   IF #Total_Waste_Volume_Percent > #Waste_Container_Interlock_Level THEN
       #Waste_Container_Interlock := TRUE;
   ELSE
       #Waste_Container_Interlock := FALSE;
   END_IF;

   IF #Total_Waste_Volume_Percent > #Waste_Container_Alarm_SP THEN
       #Waste_Container_Alarm_Level := 2;
   ELSE
       #Waste_Container_Alarm_Level := 1;
   END_IF;


   // Section commented out until ALMO system is installed
   #Alarm_Green := FALSE; // Remove when ALMO installed
   #Alarm_Red := FALSE; // Remove when ALMO installed

   (*IF #Waste_Rad_Level >= #"Waste_Rad_High-Alarm" THEN
       #Waste_Rad_Alarm := TRUE;
       #Alarm_Green := FALSE;
       #Alarm_Red := TRUE;
   ELSE
       #Waste_Rad_Alarm := FALSE;
       #Alarm_Green := TRUE;
       #Alarm_Red := FALSE;
   END_IF;*)
END_FUNCTION

FUNCTION "Total_from_Water_Supply" : Void   // FC3, SCL
{ S7_Optimized_Access := 'TRUE' }
VERSION : 0.1
   VAR_INPUT
      Removed_from_Water_Supply : Real;
      Water_Supply_Container_Size : Real;
      Water_Suppply_Interlock_Level : Real;
   END_VAR
   VAR_OUTPUT
      Total_Water_Supply : Real;
      Total_Water_Supply_Percent : Real;
      Water_Supply_Interlock : Bool;
   END_VAR
BEGIN


   #Total_Water_Supply:=#Water_Supply_Container_Size - (#Removed_from_Water_Supply/10000);
   #Total_Water_Supply_Percent := (#Total_Water_Supply / #Water_Supply_Container_Size) * 100;

   IF #Water_Suppply_Interlock_Level > #Total_Water_Supply_Percent THEN
       #Water_Supply_Interlock := TRUE;
   ELSE
       #Water_Supply_Interlock := FALSE;
   END_IF;
END_FUNCTION

FUNCTION "Convert_16bits_to_Integer" : Void   // FC4, SCL
{ S7_Optimized_Access := 'TRUE' }
VERSION : 0.1
   VAR_INPUT
      bit0 : Bool;
      bit1 : Bool;
      bit2 : Bool;
      bit3 : Bool;
      bit4 : Bool;
      bit5 : Bool;
      bit6 : Bool;
      bit7 : Bool;
      bit8 : Bool;
      bit9 : Bool;
      bit10 : Bool;
      bit11 : Bool;
      bit12 : Bool;
      bit13 : Bool;
      bit14 : Bool;
      bit15 : Bool;
   END_VAR
   VAR_OUTPUT
      Value : Int;
   END_VAR
   VAR_TEMP
      Holder : Word;
   END_VAR
BEGIN


   #Holder.%X0 := #bit0;
   #Holder.%X1 := #bit1;
   #Holder.%X2 := #bit2;
   #Holder.%X3 := #bit3;
   #Holder.%X4 := #bit4;
   #Holder.%X5 := #bit5;
   #Holder.%X6 := #bit6;
   #Holder.%X7 := #bit7;
   #Holder.%X8 := #bit8;
   #Holder.%X9 := #bit9;
   #Holder.%X10 := #bit10;
   #Holder.%X11 := #bit11;
   #Holder.%X12 := #bit12;
   #Holder.%X13 := #bit13;
   #Holder.%X14 := #bit14;
   #Holder.%X15 := #bit15;

   #Value := WORD_TO_INT(#Holder);
END_FUNCTION

FUNCTION "Pump_RPM_Conversion" : Void   // FC5, SCL
{ S7_Optimized_Access := 'TRUE' }
VERSION : 0.1
   VAR_INPUT
      Speed_SP_RPM : Real;
   END_VAR
   VAR_OUTPUT
      Speed_SP_Counts : Real;
   END_VAR
BEGIN


   #Speed_SP_Counts := 932 * #Speed_SP_RPM;
END_FUNCTION

ORGANIZATION_BLOCK "Main"   // OB1, LAD, ProgramCycle
TITLE = "Main Program Sweep (Cycle)"
{ S7_Optimized_Access := 'TRUE' }
VERSION : 0.1
   VAR_INPUT
      Initial_Call : Bool;   // Initial call of this OB
      Remanence : Bool;   // =True, if remanent data are available
   END_VAR
   VAR_TEMP
      AFI : Bool;
   END_VAR
   VAR_TEMP   // added for the SCL form of the ladder/FBD networks
      _w1 : Bool;
      _w2 : Bool;
      _w3 : Bool;
   END_VAR
BEGIN

REGION Network 1
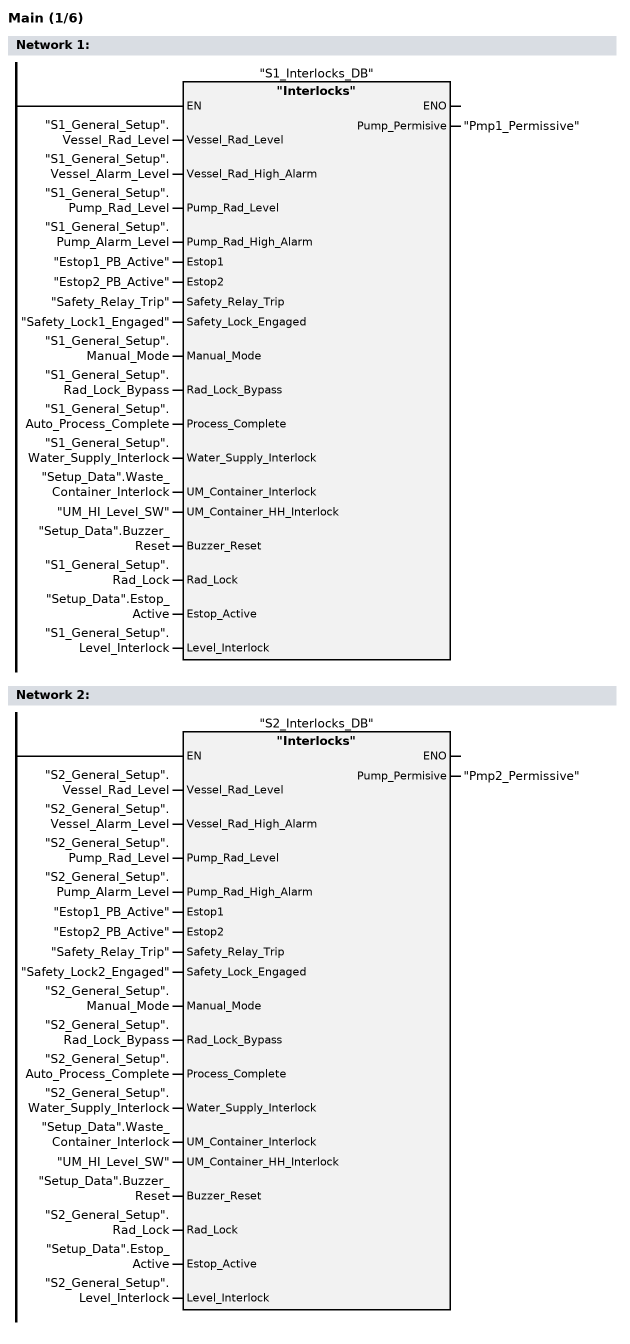
   RUNG wire#powerrail
      "S1_Interlocks_DB"(Vessel_Rad_Level := "S1_General_Setup".Vessel_Rad_Level, Vessel_Rad_High_Alarm := "S1_General_Setup".Vessel_Alarm_Level, Pump_Rad_Level := "S1_General_Setup".Pump_Rad_Level, Pump_Rad_High_Alarm := "S1_General_Setup".Pump_Alarm_Level, Estop1 := "Estop1_PB_Active", Estop2 := "Estop2_PB_Active", Safety_Relay_Trip := "Safety_Relay_Trip", Safety_Lock_Engaged := "Safety_Lock1_Engaged", Manual_Mode := "S1_General_Setup".Manual_Mode, Rad_Lock_Bypass := "S1_General_Setup".Rad_Lock_Bypass, Process_Complete := "S1_General_Setup".Auto_Process_Complete, Water_Supply_Interlock := "S1_General_Setup".Water_Supply_Interlock, UM_Container_Interlock := "Setup_Data".Waste_Container_Interlock, UM_Container_HH_Interlock := "UM_HI_Level_SW", Buzzer_Reset := "Setup_Data".Buzzer_Reset, Rad_Lock := "S1_General_Setup".Rad_Lock, Estop_Active := "Setup_Data".Estop_Active, Level_Interlock := "S1_General_Setup".Level_Interlock, Pump_Permisive => "Pmp1_Permissive")
   END_RUNG
   // the same network as SCL:
   "S1_Interlocks_DB"(Vessel_Rad_Level := "S1_General_Setup".Vessel_Rad_Level,   // "Interlocks"
                      Vessel_Rad_High_Alarm := "S1_General_Setup".Vessel_Alarm_Level,
                      Pump_Rad_Level := "S1_General_Setup".Pump_Rad_Level,
                      Pump_Rad_High_Alarm := "S1_General_Setup".Pump_Alarm_Level,
                      Estop1 := "Estop1_PB_Active",
                      Estop2 := "Estop2_PB_Active",
                      Safety_Relay_Trip := "Safety_Relay_Trip",
                      Safety_Lock_Engaged := "Safety_Lock1_Engaged",
                      Manual_Mode := "S1_General_Setup".Manual_Mode,
                      Rad_Lock_Bypass := "S1_General_Setup".Rad_Lock_Bypass,
                      Process_Complete := "S1_General_Setup".Auto_Process_Complete,
                      Water_Supply_Interlock := "S1_General_Setup".Water_Supply_Interlock,
                      UM_Container_Interlock := "Setup_Data".Waste_Container_Interlock,
                      UM_Container_HH_Interlock := "UM_HI_Level_SW",
                      Buzzer_Reset := "Setup_Data".Buzzer_Reset,
                      Rad_Lock := "S1_General_Setup".Rad_Lock,
                      Estop_Active := "Setup_Data".Estop_Active,
                      Level_Interlock := "S1_General_Setup".Level_Interlock,
                      Pump_Permisive => "Pmp1_Permissive");
END_REGION

REGION Network 2
   RUNG wire#powerrail
      "S2_Interlocks_DB"(Vessel_Rad_Level := "S2_General_Setup".Vessel_Rad_Level, Vessel_Rad_High_Alarm := "S2_General_Setup".Vessel_Alarm_Level, Pump_Rad_Level := "S2_General_Setup".Pump_Rad_Level, Pump_Rad_High_Alarm := "S2_General_Setup".Pump_Alarm_Level, Estop1 := "Estop1_PB_Active", Estop2 := "Estop2_PB_Active", Safety_Relay_Trip := "Safety_Relay_Trip", Safety_Lock_Engaged := "Safety_Lock2_Engaged", Manual_Mode := "S2_General_Setup".Manual_Mode, Rad_Lock_Bypass := "S2_General_Setup".Rad_Lock_Bypass, Process_Complete := "S2_General_Setup".Auto_Process_Complete, Water_Supply_Interlock := "S2_General_Setup".Water_Supply_Interlock, UM_Container_Interlock := "Setup_Data".Waste_Container_Interlock, UM_Container_HH_Interlock := "UM_HI_Level_SW", Buzzer_Reset := "Setup_Data".Buzzer_Reset, Rad_Lock := "S2_General_Setup".Rad_Lock, Estop_Active := "Setup_Data".Estop_Active, Level_Interlock := "S2_General_Setup".Level_Interlock, Pump_Permisive => "Pmp2_Permissive")
   END_RUNG
   // the same network as SCL:
   "S2_Interlocks_DB"(Vessel_Rad_Level := "S2_General_Setup".Vessel_Rad_Level,   // "Interlocks"
                      Vessel_Rad_High_Alarm := "S2_General_Setup".Vessel_Alarm_Level,
                      Pump_Rad_Level := "S2_General_Setup".Pump_Rad_Level,
                      Pump_Rad_High_Alarm := "S2_General_Setup".Pump_Alarm_Level,
                      Estop1 := "Estop1_PB_Active",
                      Estop2 := "Estop2_PB_Active",
                      Safety_Relay_Trip := "Safety_Relay_Trip",
                      Safety_Lock_Engaged := "Safety_Lock2_Engaged",
                      Manual_Mode := "S2_General_Setup".Manual_Mode,
                      Rad_Lock_Bypass := "S2_General_Setup".Rad_Lock_Bypass,
                      Process_Complete := "S2_General_Setup".Auto_Process_Complete,
                      Water_Supply_Interlock := "S2_General_Setup".Water_Supply_Interlock,
                      UM_Container_Interlock := "Setup_Data".Waste_Container_Interlock,
                      UM_Container_HH_Interlock := "UM_HI_Level_SW",
                      Buzzer_Reset := "Setup_Data".Buzzer_Reset,
                      Rad_Lock := "S2_General_Setup".Rad_Lock,
                      Estop_Active := "Setup_Data".Estop_Active,
                      Level_Interlock := "S2_General_Setup".Level_Interlock,
                      Pump_Permisive => "Pmp2_Permissive");
END_REGION

REGION Network 3
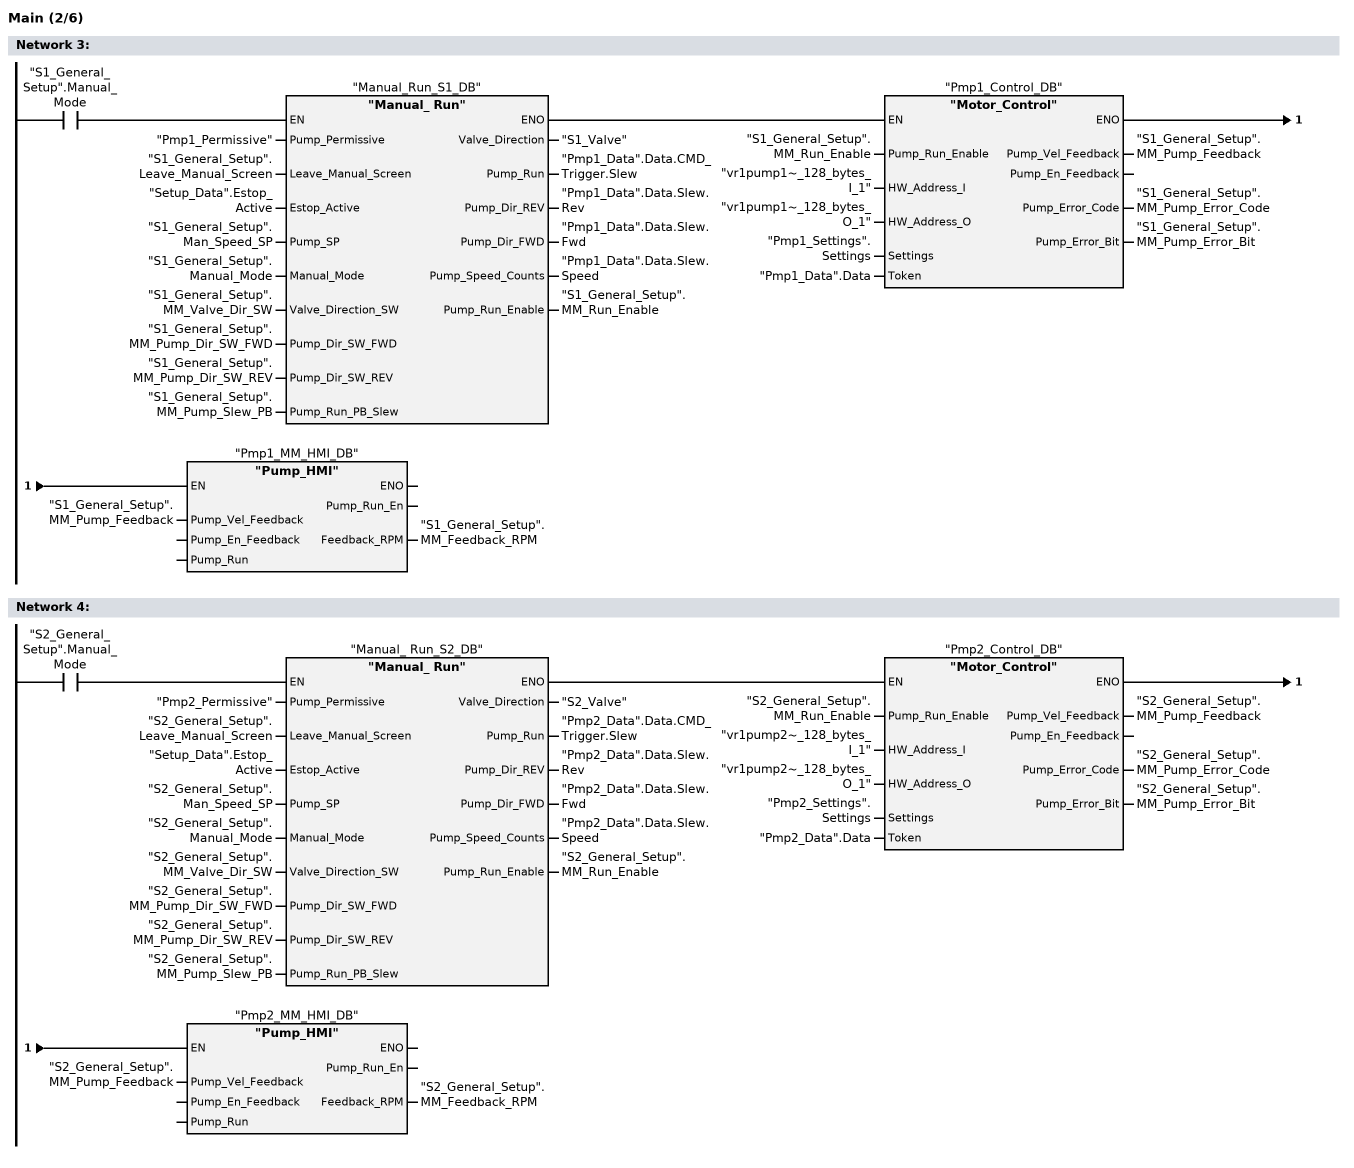
   RUNG wire#powerrail
      Contact( "S1_General_Setup".Manual_Mode )
      "Manual_Run_S1_DB"(Pump_Permissive := "Pmp1_Permissive", Leave_Manual_Screen := "S1_General_Setup".Leave_Manual_Screen, Estop_Active := "Setup_Data".Estop_Active, Pump_SP := "S1_General_Setup".Man_Speed_SP, Manual_Mode := "S1_General_Setup".Manual_Mode, Valve_Direction_SW := "S1_General_Setup".MM_Valve_Dir_SW, Pump_Dir_SW_FWD := "S1_General_Setup".MM_Pump_Dir_SW_FWD, Pump_Dir_SW_REV := "S1_General_Setup".MM_Pump_Dir_SW_REV, Pump_Run_PB_Slew := "S1_General_Setup".MM_Pump_Slew_PB, Valve_Direction => "S1_Valve", Pump_Run => "Pmp1_Data".Data.CMD_Trigger.Slew, Pump_Dir_REV => "Pmp1_Data".Data.Slew.Rev, Pump_Dir_FWD => "Pmp1_Data".Data.Slew.Fwd, Pump_Speed_Counts => "Pmp1_Data".Data.Slew.Speed, Pump_Run_Enable => "S1_General_Setup".MM_Run_Enable)
      "Pmp1_Control_DB"(Pump_Run_Enable := "S1_General_Setup".MM_Run_Enable, HW_Address_I := "vr1pump1~_128_bytes_I_1", HW_Address_O := "vr1pump1~_128_bytes_O_1", Settings := "Pmp1_Settings".Settings, Token := "Pmp1_Data".Data, Pump_Vel_Feedback => "S1_General_Setup".MM_Pump_Feedback, Pump_En_Feedback =>, Pump_Error_Code => "S1_General_Setup".MM_Pump_Error_Code, Pump_Error_Bit => "S1_General_Setup".MM_Pump_Error_Bit)
      "Pmp1_MM_HMI_DB"(Pump_Vel_Feedback := "S1_General_Setup".MM_Pump_Feedback, Pump_En_Feedback :=, Pump_Run :=, Pump_Run_En =>, Feedback_RPM => "S1_General_Setup".MM_Feedback_RPM)
   END_RUNG
   // the same network as SCL:
   "Manual_Run_S1_DB"(EN := "S1_General_Setup".Manual_Mode,   // "Manual_ Run"
                      Pump_Permissive := "Pmp1_Permissive",
                      Leave_Manual_Screen := "S1_General_Setup".Leave_Manual_Screen,
                      Estop_Active := "Setup_Data".Estop_Active,
                      Pump_SP := "S1_General_Setup".Man_Speed_SP,
                      Manual_Mode := "S1_General_Setup".Manual_Mode,
                      Valve_Direction_SW := "S1_General_Setup".MM_Valve_Dir_SW,
                      Pump_Dir_SW_FWD := "S1_General_Setup".MM_Pump_Dir_SW_FWD,
                      Pump_Dir_SW_REV := "S1_General_Setup".MM_Pump_Dir_SW_REV,
                      Pump_Run_PB_Slew := "S1_General_Setup".MM_Pump_Slew_PB,
                      Valve_Direction => "S1_Valve",
                      Pump_Run => "Pmp1_Data".Data.CMD_Trigger.Slew,
                      Pump_Dir_REV => "Pmp1_Data".Data.Slew.Rev,
                      Pump_Dir_FWD => "Pmp1_Data".Data.Slew.Fwd,
                      Pump_Speed_Counts => "Pmp1_Data".Data.Slew.Speed,
                      Pump_Run_Enable => "S1_General_Setup".MM_Run_Enable,
                      ENO => #_w1);
   "Pmp1_Control_DB"(EN := #_w1,   // "Motor_Control"
                     Pump_Run_Enable := "S1_General_Setup".MM_Run_Enable,
                     HW_Address_I := "vr1pump1~_128_bytes_I_1",
                     HW_Address_O := "vr1pump1~_128_bytes_O_1",
                     Settings := "Pmp1_Settings".Settings,
                     Token := "Pmp1_Data".Data,
                     Pump_Vel_Feedback => "S1_General_Setup".MM_Pump_Feedback,
                     Pump_Error_Code => "S1_General_Setup".MM_Pump_Error_Code,
                     Pump_Error_Bit => "S1_General_Setup".MM_Pump_Error_Bit,
                     ENO => #_w2);
   IF #_w2 THEN
       "Pmp1_MM_HMI_DB"(Pump_Vel_Feedback := "S1_General_Setup".MM_Pump_Feedback,   // "Pump_HMI"
                        Feedback_RPM => "S1_General_Setup".MM_Feedback_RPM);
   END_IF;
END_REGION

REGION Network 4
   RUNG wire#powerrail
      Contact( "S2_General_Setup".Manual_Mode )
      "Manual_ Run_S2_DB"(Pump_Permissive := "Pmp2_Permissive", Leave_Manual_Screen := "S2_General_Setup".Leave_Manual_Screen, Estop_Active := "Setup_Data".Estop_Active, Pump_SP := "S2_General_Setup".Man_Speed_SP, Manual_Mode := "S2_General_Setup".Manual_Mode, Valve_Direction_SW := "S2_General_Setup".MM_Valve_Dir_SW, Pump_Dir_SW_FWD := "S2_General_Setup".MM_Pump_Dir_SW_FWD, Pump_Dir_SW_REV := "S2_General_Setup".MM_Pump_Dir_SW_REV, Pump_Run_PB_Slew := "S2_General_Setup".MM_Pump_Slew_PB, Valve_Direction => "S2_Valve", Pump_Run => "Pmp2_Data".Data.CMD_Trigger.Slew, Pump_Dir_REV => "Pmp2_Data".Data.Slew.Rev, Pump_Dir_FWD => "Pmp2_Data".Data.Slew.Fwd, Pump_Speed_Counts => "Pmp2_Data".Data.Slew.Speed, Pump_Run_Enable => "S2_General_Setup".MM_Run_Enable)
      "Pmp2_Control_DB"(Pump_Run_Enable := "S2_General_Setup".MM_Run_Enable, HW_Address_I := "vr1pump2~_128_bytes_I_1", HW_Address_O := "vr1pump2~_128_bytes_O_1", Settings := "Pmp2_Settings".Settings, Token := "Pmp2_Data".Data, Pump_Vel_Feedback => "S2_General_Setup".MM_Pump_Feedback, Pump_En_Feedback =>, Pump_Error_Code => "S2_General_Setup".MM_Pump_Error_Code, Pump_Error_Bit => "S2_General_Setup".MM_Pump_Error_Bit)
      "Pmp2_MM_HMI_DB"(Pump_Vel_Feedback := "S2_General_Setup".MM_Pump_Feedback, Pump_En_Feedback :=, Pump_Run :=, Pump_Run_En =>, Feedback_RPM => "S2_General_Setup".MM_Feedback_RPM)
   END_RUNG
   // the same network as SCL:
   "Manual_ Run_S2_DB"(EN := "S2_General_Setup".Manual_Mode,   // "Manual_ Run"
                       Pump_Permissive := "Pmp2_Permissive",
                       Leave_Manual_Screen := "S2_General_Setup".Leave_Manual_Screen,
                       Estop_Active := "Setup_Data".Estop_Active,
                       Pump_SP := "S2_General_Setup".Man_Speed_SP,
                       Manual_Mode := "S2_General_Setup".Manual_Mode,
                       Valve_Direction_SW := "S2_General_Setup".MM_Valve_Dir_SW,
                       Pump_Dir_SW_FWD := "S2_General_Setup".MM_Pump_Dir_SW_FWD,
                       Pump_Dir_SW_REV := "S2_General_Setup".MM_Pump_Dir_SW_REV,
                       Pump_Run_PB_Slew := "S2_General_Setup".MM_Pump_Slew_PB,
                       Valve_Direction => "S2_Valve",
                       Pump_Run => "Pmp2_Data".Data.CMD_Trigger.Slew,
                       Pump_Dir_REV => "Pmp2_Data".Data.Slew.Rev,
                       Pump_Dir_FWD => "Pmp2_Data".Data.Slew.Fwd,
                       Pump_Speed_Counts => "Pmp2_Data".Data.Slew.Speed,
                       Pump_Run_Enable => "S2_General_Setup".MM_Run_Enable,
                       ENO => #_w1);
   "Pmp2_Control_DB"(EN := #_w1,   // "Motor_Control"
                     Pump_Run_Enable := "S2_General_Setup".MM_Run_Enable,
                     HW_Address_I := "vr1pump2~_128_bytes_I_1",
                     HW_Address_O := "vr1pump2~_128_bytes_O_1",
                     Settings := "Pmp2_Settings".Settings,
                     Token := "Pmp2_Data".Data,
                     Pump_Vel_Feedback => "S2_General_Setup".MM_Pump_Feedback,
                     Pump_Error_Code => "S2_General_Setup".MM_Pump_Error_Code,
                     Pump_Error_Bit => "S2_General_Setup".MM_Pump_Error_Bit,
                     ENO => #_w2);
   IF #_w2 THEN
       "Pmp2_MM_HMI_DB"(Pump_Vel_Feedback := "S2_General_Setup".MM_Pump_Feedback,   // "Pump_HMI"
                        Feedback_RPM => "S2_General_Setup".MM_Feedback_RPM);
   END_IF;
END_REGION

